# B&R Automation Studio project PT_KB_V01 (part 9)

#### Cyclic.st - Cyclic code
```iecst
PROGRAM _CYCLIC
	(* ======================================================================== *)
	(* Rad_PG_KB_CYCLIC                                                          *)
	(* Rad_PG_KB.Sequence.State masina izbora i rada izvora termalne vode: BRB2 (1) ili IEBKB1 (2). *)
	(* Prelazak izmedju grana ide iskljucivo preko PG_00_Stand_By - direktan     *)
	(* prelazak 1->2 ili 2->1 nije moguc.                                       *)
	(* ======================================================================== *)

	(* -------------------------------------------------------------------------- *)
	(* 1) Vracanje projektnih podrazumevanih parametara                          *)
	(* -------------------------------------------------------------------------- *)
	IF Rad_PG_KB.HMI.Cntrl.SetDefaultParameters THEN
		(* 1.1) Izlazne pumpe iza prihvatnog tanka. *)
		(* Aktivni SP zavisi od izabrane regulacije pritiska ili nivoa. *)
		PGRad.Par.SetPritisakPotisa := 1.2;
		PGRad.Par.SetPointNivoTanka := 1.5;
		PGRad.Par.SetPointNivoTankaUpozorenje := 2.1; (* Informativni prag; stvarni fizicki preliv je ~2.15-2.2 m. *)
		PGRad.Par.PocetnaFrekvencaIzlaznePumpe := 10.0;

		(* Centralne granice PID izlaza za obe pumpe iza prihvatnog tanka. *)
		PGRad.Par.MinFR_Pumpe := 10.0;
		PGRad.Par.MaxFR_Pumpe := 45.0;
		(* MinFR_Pumpe se u PID_Pu_PT propagira na PID_Pu_PT.MinOut. *)
		(* MaxFR_Pumpe se preko PGRad_Cmd.PID.MaxOut propagira na PID_Pu_PT.MaxOut. *)
		PGRad.Par.TimeSP.OverlapPumpi_s := 10.0;
		PGRad.Par.TimeSP.AutoRestartDelay_s := 60.0;

		(* 1.2) BRB2 priprema i ispiranje dovodne grane. *)
		PGRad.Par.MinProtok := 1.5; (* Rezervisano; trenutno nema izvrsnog potrosaca. *)
		PGRad.Par.MaxProtok := 16.2;
		PGRad.Par.SetPointMinTempIspiranja := 60.0;
		PGRad.Par.BRB2Preparation.MinTemperature_degC := 60.0;
		PGRad.Par.BRB2Preparation.MinFlow_lps := 3.0;
		PGRad.Par.BRB2Preparation.FlowTimeout_s := 30.0;
		PGRad.Par.BRB2Preparation.TemperatureAlarm_s := 5400.0;
		PGRad.Par.BRB2Preparation.TemperatureStopDelay_s := 900.0;
		PGRad.Par.BRB2Preparation.PressureAlarmDelay_s := 5.0;
		PGRad.Par.BRB2Preparation.PressureStopDelay_s := 8.0;

		(* 1.3) Lokalna hidraulika PV05 i ulaza u prihvatni tank. *)
		PGRad.Par.SetPointPritisakPV05Ispiranje := 5.5;
		PGRad.Par.SetPointPritisakUlazTanka := 5.5;
		PGRad.Par.SetPointMaxPritisakDolaznaCev := 6.5;
		PGRad.Par.TimeSP.PrelazPV05Cuvar_s := 15.0;
		PGRad.Par.MaxOtvorPropZaZatvaranje := 3;

		(* 1.4) Kontrolisani transfer sa IEBKB1 na BRB2. *)
		PGRad.Par.Transfer.PV05StartPressure_bar := 5.5;
		PGRad.Par.Transfer.PV05FinalPressure_bar := 6.5;
		PGRad.Par.Transfer.TankInletPressure_bar := 5.5;
		PGRad.Par.Transfer.PressureRamp_s := 15.0;
		PGRad.Par.Transfer.FlowTimeout_s := 30.0;
		PGRad.Par.Transfer.PV05ClosedPercent := 4.0;

		(* 1.5) Zajednicki nadzor ventila i procesnih interlock-a. *)
		PGRad.Par.TimeSP.ValvePositionTimeout_s := 30.0;
		PGRad.Par.TimeSP.InterlockDebounce_s := 2.0;

		(* 1.6) BRB2 odzracivanje: oba ventila, prag 1.5 bar sa 0.5 bar histerezom. *)
		PGRad.Par.AirRelease.BRB2.PV03.NumberOfLS := 2;
		PGRad.Par.AirRelease.BRB2.PV03.PressureSP_bar := 1.5;
		PGRad.Par.AirRelease.BRB2.PV03.PressureHysteresis_bar := 0.5;
		PGRad.Par.AirRelease.BRB2.PV03.LS1.SP_Percent := 20.0;
		PGRad.Par.AirRelease.BRB2.PV03.LS1.Ramp_PercentPerSecond := 2.0;
		PGRad.Par.AirRelease.BRB2.PV03.LS1.ConfirmTime_s := 1.0;
		PGRad.Par.AirRelease.BRB2.PV03.LS2.SP_Percent := 89.0;
		PGRad.Par.AirRelease.BRB2.PV03.LS2.Ramp_PercentPerSecond := 15.0;
		PGRad.Par.AirRelease.BRB2.PV03.LS2.ConfirmTime_s := 1.0;
		PGRad.Par.AirRelease.BRB2.PV04 := PGRad.Par.AirRelease.BRB2.PV03;

		(* 1.7) IEBKB1 odzracivanje: aktivan je PV03 sa nizim pragom pritiska. *)
		PGRad.Par.AirRelease.IEBKB1.PV03.NumberOfLS := 2;
		PGRad.Par.AirRelease.IEBKB1.PV03.PressureSP_bar := 0.15;
		PGRad.Par.AirRelease.IEBKB1.PV03.PressureHysteresis_bar := 0.05;
		PGRad.Par.AirRelease.IEBKB1.PV03.LS1.SP_Percent := 20.0;
		PGRad.Par.AirRelease.IEBKB1.PV03.LS1.Ramp_PercentPerSecond := 2.0;
		PGRad.Par.AirRelease.IEBKB1.PV03.LS1.ConfirmTime_s := 1.0;
		PGRad.Par.AirRelease.IEBKB1.PV03.LS2.SP_Percent := 89.0;
		PGRad.Par.AirRelease.IEBKB1.PV03.LS2.Ramp_PercentPerSecond := 15.0;
		PGRad.Par.AirRelease.IEBKB1.PV03.LS2.ConfirmTime_s := 1.0;
		PGRad.Par.AirRelease.IEBKB1.PV04 := PGRad.Par.AirRelease.IEBKB1.PV03;

		Rad_PG_KB.HMI.Cntrl.SetDefaultParameters := FALSE;
	END_IF

	(* -------------------------------------------------------------------------- *)
	(* 2) Podrazumevane neretentivne komande po scan-u                            *)
	(* -------------------------------------------------------------------------- *)
	PGRad_Cmd.Aktivan := FALSE;
	PGRad_Cmd.Ventili._03_Open := FALSE;
	PGRad_Cmd.Ventili._04_Open := FALSE;
	PGRad_Cmd.Ventili._05_Open := FALSE;
	PGRad_Cmd.Ventili._06_Open := FALSE;
	PGRad_Cmd.Ventili._07_Open := FALSE;

	PGRad_Cmd.PropVentili.PV01.Enable := FALSE;
	PGRad_Cmd.PropVentili.PV01.SP_Percent := 0.0;
	PGRad_Cmd.PropVentili.PV02.Enable := FALSE;
	PGRad_Cmd.PropVentili.PV02.SP_Percent := 0.0;
	PGRad_Cmd.PropVentili.PV05.Enable := FALSE;
	PGRad_Cmd.PropVentili.PV05.SP_Percent := 0.0;
	PGRad_Cmd.AirRelease.PV03.Enable := FALSE;
	PGRad_Cmd.AirRelease.PV04.Enable := FALSE;
	PGRad_Cmd.AirRelease.UseIEBKB1Parameters := FALSE;
	PGRad_Cmd.AirRelease.ResetAll := Rad_PG_KB.HMI.Cntrl.Reset;

	PGRad_Cmd.Pumpe._01.Run := FALSE;
	PGRad_Cmd.Pumpe._02.Run := FALSE;
	PGRad_Cmd.PID.Enable := FALSE;
	PGRad_Cmd.PID.ActValue := 0.0;
	PGRad_Cmd.PID.SetValue := 0.0;
	PGRad_Cmd.PID.Invert := FALSE;
	(* Jedinstvena maksimalna PID frekvencija ne zavisi od izabrane pumpe. *)
	PGRad_Cmd.PID.MaxOut := PGRad.Par.MaxFR_Pumpe;
	PGRad_Cmd.PID.EnableTracking := FALSE;
	(* Jedinstvena pocetna frekvencija koristi se pri ukljucenju PID tracking-a. *)
	PGRad_Cmd.PID.TrackingValue := PGRad.Par.PocetnaFrekvencaIzlaznePumpe;
	PGRad_BRB2Cmd.RadKaPodstanici := FALSE;
	PGRad_BRB2Cmd.ZahtevStarta := FALSE;
	PGRad_BRB2Cmd.ZahtevZaustavljanja := FALSE;
	PGRad_BRB2Cmd.ManualMode := Rad_PG_KB.HMI.Manual.Enable;
	PGRad_BRB2Cmd.ManualSequence := Rad_PG_KB.HMI.Manual.Sequence;
	PGRad_BRB2Cmd.ManualStart := Rad_PG_KB.HMI.Manual.Start;
	PGRad_BRB2Cmd.ManualStop := Rad_PG_KB.HMI.Manual.Stop;
	PGRad_BRB2Cmd.ManualNextStep := Rad_PG_KB.HMI.Manual.NextStep;
	PGRad_BRB2Cmd.ManualAbort := Rad_PG_KB.HMI.Manual.Abort;
	PGRad_BRB2Cmd.VentiliPodstaniceZatvoreni := FALSE;
	PGRad_BRB2Cmd.PritisakIEBKB1 := IEB_KB1.Sens.Pt.B_02._01_value;
	PGRad_BRB2Cmd.PodstanicaURezimuRada := FALSE;
	PGRad_BRB2Cmd.RegulationMode := 0;
	PGRad_BRB2Cmd.RegulationPV := 0.0;
	PGRad_BRB2Cmd.RegulationSP := 0.0;
	PGRad_BRB2Cmd.RegulationPVValid := FALSE;
	PGRad_BRB2Cmd.RegulationInvert := FALSE;
	PGRad_BRB2Cmd.NivoPrihvatniSud := NivoPrihvatniSud;
	IEB_KB1.Cntrl.Comm.Podstanica.Zahtev.ZahtevVode := FALSE;
	IEB_KB1.Cntrl.Comm.Podstanica.Zahtev.NivoPrihvatnogTanka := NivoPrihvatniSud;
	IEB_KB1.Cntrl.Comm.Podstanica.Zahtev.CiljaniProtok := PGRad.Par.MaxProtok;
	IEB_KB1.Cntrl.Comm.Podstanica.Zahtev.ModRada := 0;
	IEB_KB1.Cntrl.proba := FALSE;

	(* Izbor izvora sa HMI prihvata se samo u bezbednom Standby stanju. *)
	IF Rad_PG_KB.Sequence.State = PG_00_Stand_By THEN
		IF Rad_PG_KB.HMI.Cntrl.SelectIEBKB1 THEN
			PGRad.Ctrl.SelektovaniIzvor := _02_IEBKB1;
		ELSE
			PGRad.Ctrl.SelektovaniIzvor := _01_BRB2;
		END_IF;
	ELSE
		Rad_PG_KB.HMI.Cntrl.SelectIEBKB1 := PGRad.Ctrl.SelektovaniIzvor = _02_IEBKB1;
	END_IF;

	(* -------------------------------------------------------------------------- *)
	(* 3) Tajmeri pripreme BRB2 dovodne putanje                                  *)
	(* -------------------------------------------------------------------------- *)
	Rad_PG_KB.Timer.PG_V01.Close.IN := FALSE;
	Rad_PG_KB.Timer.PG_V01.Close.PT := REAL_TO_TIME(PGRad.Par.TimeSP.ValvePositionTimeout_s * 1000.0);
	Rad_PG_KB.Timer.PG_V02.Open.IN := FALSE;
	Rad_PG_KB.Timer.PG_V02.Open.PT := REAL_TO_TIME(PGRad.Par.TimeSP.ValvePositionTimeout_s * 1000.0);
	Rad_PG_KB.Timer.PG_V02.Close.IN := FALSE;
	Rad_PG_KB.Timer.PG_V02.Close.PT := REAL_TO_TIME(PGRad.Par.TimeSP.ValvePositionTimeout_s * 1000.0);
	Rad_PG_KB.Timer.PG_V01.Open.IN := FALSE;
	Rad_PG_KB.Timer.PG_V01.Open.PT := REAL_TO_TIME(PGRad.Par.TimeSP.ValvePositionTimeout_s * 1000.0);
	Rad_PG_KB.Timer.IEBKB1.StartProtokTimeout.IN := FALSE;
	Rad_PG_KB.Timer.IEBKB1.StartProtokTimeout.PT := REAL_TO_TIME(PGRad.Par.TimeSP.ValvePositionTimeout_s * 1000.0);
	Rad_PG_KB.Timer.IEBKB1.ProtokNula.IN := FALSE;
	Rad_PG_KB.Timer.IEBKB1.ProtokNula.PT := REAL_TO_TIME(PGRad.Par.TimeSP.InterlockDebounce_s * 1000.0);
	Rad_PG_KB.Timer.IEBKB1.StopProtokTimeout.IN := FALSE;
	Rad_PG_KB.Timer.IEBKB1.StopProtokTimeout.PT := REAL_TO_TIME(PGRad.Par.TimeSP.ValvePositionTimeout_s * 1000.0);
	Rad_PG_KB.Timer.PG_V05.Close.IN := FALSE;
	Rad_PG_KB.Timer.PG_V05.Close.PT := REAL_TO_TIME(PGRad.Par.TimeSP.ValvePositionTimeout_s * 1000.0);
	Rad_PG_KB.Timer.Transfer.PV05Guard.IN := FALSE;
	Rad_PG_KB.Timer.Transfer.PV05Guard.PT := REAL_TO_TIME(PGRad.Par.TimeSP.PrelazPV05Cuvar_s * 1000.0);
	Rad_PG_KB.Timer.BRB2.PreparationFlow.IN := FALSE;
	Rad_PG_KB.Timer.BRB2.PreparationFlow.PT := REAL_TO_TIME(PGRad.Par.BRB2Preparation.FlowTimeout_s * 1000.0);
	Rad_PG_KB.Timer.BRB2.TemperatureAlarm.IN := FALSE;
	Rad_PG_KB.Timer.BRB2.TemperatureAlarm.PT := REAL_TO_TIME(PGRad.Par.BRB2Preparation.TemperatureAlarm_s * 1000.0);
	Rad_PG_KB.Timer.BRB2.TemperatureStop.IN := FALSE;
	Rad_PG_KB.Timer.BRB2.TemperatureStop.PT := REAL_TO_TIME(PGRad.Par.BRB2Preparation.TemperatureStopDelay_s * 1000.0);
	Rad_PG_KB.Timer.BRB2.PressureAlarm.IN := FALSE;
	Rad_PG_KB.Timer.BRB2.PressureAlarm.PT := REAL_TO_TIME(PGRad.Par.BRB2Preparation.PressureAlarmDelay_s * 1000.0);
	Rad_PG_KB.Timer.BRB2.PressureStop.IN := FALSE;
	Rad_PG_KB.Timer.BRB2.PressureStop.PT := REAL_TO_TIME(PGRad.Par.BRB2Preparation.PressureStopDelay_s * 1000.0);
	Rad_PG_KB.Timer.Transfer.Flow.IN := FALSE;
	Rad_PG_KB.Timer.Transfer.Flow.PT := REAL_TO_TIME(PGRad.Par.Transfer.FlowTimeout_s * 1000.0);
	Rad_PG_KB.AutoRestart.Timer.IN := FALSE;
	Rad_PG_KB.AutoRestart.Timer.PT := REAL_TO_TIME(PGRad.Par.TimeSP.AutoRestartDelay_s * 1000.0);

	(* -------------------------------------------------------------------------- *)
	(* 3b) Informativna napomena: nivo prihvatnog suda blizu fizickog preliva.    *)
	(* Samo obavestenje za HMI, bez ikakve upravljacke akcije ili interlock-a -   *)
	(* ocekivano tokom regulacije temperature sekundara/protoka sa bunara uz      *)
	(* pritisak potisa izlazne pumpe.                                            *)
	(* -------------------------------------------------------------------------- *)
	Rad_PG_KB.Status.PrihvatniSudBlizuPreliva := NivoPrihvatniSud >= PGRad.Par.SetPointNivoTankaUpozorenje;

	(* -------------------------------------------------------------------------- *)
	(* 4) Glavna state masina izvora termalne vode                                *)
	(* -------------------------------------------------------------------------- *)
	(* Rad_PG_KB.HMI.Manual.Start grane imaju prioritet evaluacije. BRB2 auto-start je blokiran  *)
	(* sa Rad_PG_KB.HMI.Manual.Enable, dok IEBKB1 auto-start grana nema eksplicitnu tu proveru.    *)
	CASE Rad_PG_KB.Sequence.State OF

		PG_00_Stand_By:
			(* Neretentivni vektor je bezbedno resetovan u sekciji 2; V01/V02 se ne menjaju. *)
			Rad_PG_KB.Status.PV05.FlushingOpened := FALSE;
			(* Automatski start posle WARMSTART-a (nestanak struje), samo ako je operater *)
			(* aktivirao PGRad.Ctrl.AutoRestart. Prekida se ako se pojavi Fault ili se    *)
			(* rucno napusti Standby/automatski rezim u toku odlozenog starta.           *)
			Rad_PG_KB.AutoRestart.Timer.IN :=
				Rad_PG_KB.AutoRestart.WarmstartDetected
				AND PGRad.Ctrl.AutoRestart
				AND (NOT Rad_PG_KB.HMI.Manual.Enable)
				AND (NOT Rad_PG_KB.Diag.Fault.Latched)
				AND (PGRad.Ctrl.RegulacionaVarijanta <> _00_neaktivan);
			IF Rad_PG_KB.AutoRestart.Timer.Q THEN
				Rad_PG_KB.HMI.Cntrl.Start := TRUE;
				Rad_PG_KB.AutoRestart.WarmstartDetected := FALSE; (* jednokratno okidanje *)
			END_IF;
			(* Start je dozvoljen samo sa izabranim izvorom i regulacionom varijantom. *)
			IF Rad_PG_KB.HMI.Manual.Enable AND Rad_PG_KB.HMI.Manual.Start AND (Rad_PG_KB.HMI.Manual.Sequence = 1) THEN
				PGRad.Ctrl.SelektovaniIzvor := _01_BRB2;
				Rad_PG_KB.HMI.Manual.Start := FALSE;
				Rad_PG_KB.Sequence.State := PG_01_Priprema_BRB2;
				Rad_PG_KB.Sequence.Substep := 0;
			ELSIF Rad_PG_KB.HMI.Manual.Enable AND Rad_PG_KB.HMI.Manual.Start AND (Rad_PG_KB.HMI.Manual.Sequence = 2) THEN
				PGRad.Ctrl.SelektovaniIzvor := _02_IEBKB1;
				Rad_PG_KB.HMI.Manual.Start := FALSE;
				Rad_PG_KB.Sequence.State := PG_11_Priprema_IEBKB1;
				Rad_PG_KB.Sequence.Substep := 0;
			ELSIF Rad_PG_KB.HMI.Cntrl.Start
				AND (NOT Rad_PG_KB.HMI.Manual.Enable)
				AND (NOT Rad_PG_KB.Diag.Fault.Latched)
				AND (PGRad.Ctrl.RegulacionaVarijanta <> _00_neaktivan)
				AND (PGRad.Ctrl.SelektovaniIzvor = _01_BRB2) THEN
				Rad_PG_KB.Sequence.State := PG_01_Priprema_BRB2;
				Rad_PG_KB.Sequence.Substep := 0;
			ELSIF Rad_PG_KB.HMI.Cntrl.Start
				AND (NOT Rad_PG_KB.Diag.Fault.Latched)
				AND (PGRad.Ctrl.RegulacionaVarijanta <> _00_neaktivan)
				AND (PGRad.Ctrl.SelektovaniIzvor = _02_IEBKB1) THEN
				Rad_PG_KB.Sequence.State := PG_11_Priprema_IEBKB1;
				Rad_PG_KB.Sequence.Substep := 0;
			END_IF

		PG_01_Priprema_BRB2:
			IF Rad_PG_KB.HMI.Manual.Stop OR Rad_PG_KB.HMI.Manual.Abort THEN
				Rad_PG_KB.HMI.Cntrl.Stop := TRUE;
				Rad_PG_KB.HMI.Manual.Stop := FALSE;
				Rad_PG_KB.HMI.Manual.Abort := FALSE;
			END_IF;
			PGRad_BRB2Cmd.RadKaPodstanici := TRUE;
			PGRad_BRB2Cmd.ZahtevStarta := TRUE;
			CASE Rad_PG_KB.Sequence.Substep OF
				0:
					(* Prioritet BRB2: najpre zatvori dovod sa IEBKB1. *)
					PGRad.CmdRetain.V01_Open := FALSE;
					Rad_PG_KB.Sequence.Substep := 1;

				1:
					(* Otvaranje BRB2 dovoda je dozvoljeno tek po potvrdi zatvorenog V01. *)
					PGRad.CmdRetain.V01_Open := FALSE;
					Rad_PG_KB.Timer.PG_V01.Close.IN := NOT PG.Act.AV._1.Closed;
					IF PG.Act.AV._1.Closed AND (NOT Rad_PG_KB.HMI.Manual.Enable OR Rad_PG_KB.HMI.Manual.NextStep) THEN
						Rad_PG_KB.HMI.Manual.NextStep := FALSE;
						PGRad.CmdRetain.V02_Open := TRUE;
						Rad_PG_KB.Sequence.Substep := 2;
					ELSIF Rad_PG_KB.Timer.PG_V01.Close.Q THEN
						PGRad.CmdRetain.V01_Open := FALSE;
						PGRad.CmdRetain.V02_Open := FALSE;
						Rad_PG_KB.Diag.Fault.Latched := TRUE;
						Rad_PG_KB.Diag.Fault.Code := 11;
						Rad_PG_KB.Diag.Fault.Text := 'PG_V01 nije zatvoren za zadato vreme';
						Rad_PG_KB.Sequence.State := PG_00_Stand_By;
						Rad_PG_KB.Sequence.Substep := 0;
					END_IF

				2:
					(* Ceka se fizicka potvrda otvorenog BRB2 dovoda. *)
					PGRad.CmdRetain.V01_Open := FALSE;
					PGRad.CmdRetain.V02_Open := TRUE;
					Rad_PG_KB.Timer.PG_V02.Open.IN := NOT PG.Act.AV._2.Opened;
					IF PG.Act.AV._2.Opened AND (NOT Rad_PG_KB.HMI.Manual.Enable OR Rad_PG_KB.HMI.Manual.NextStep) THEN
						Rad_PG_KB.HMI.Manual.NextStep := FALSE;
						Rad_PG_KB.Sequence.Substep := 3;
					ELSIF Rad_PG_KB.Timer.PG_V02.Open.Q THEN
						PGRad.CmdRetain.V01_Open := FALSE;
						PGRad.CmdRetain.V02_Open := FALSE;
						Rad_PG_KB.Diag.Fault.Latched := TRUE;
						Rad_PG_KB.Diag.Fault.Code := 12;
						Rad_PG_KB.Diag.Fault.Text := 'PG_V02 nije otvoren za zadato vreme';
						Rad_PG_KB.Sequence.State := PG_00_Stand_By;
						Rad_PG_KB.Sequence.Substep := 0;
					END_IF

				3:
					(* PG_PV05 se otvara nakon dostignutog PT06 pritiska; temperatura se proverava tek posle BRB2 minimuma. *)
					IF PG.Sens.Pt._6.AI_Output.ScaledValue >= PGRad.Par.SetPointPritisakPV05Ispiranje THEN
						Rad_PG_KB.Status.PV05.FlushingOpened := TRUE;
					END_IF;
					IF Rad_PG_KB.Status.PV05.FlushingOpened THEN
						PGRad_Cmd.Aktivan := TRUE;
						PGRad_Cmd.PropVentili.PV05.Enable := TRUE;
					END_IF;
					IF PGRad_BRB2.IspiranjeMinTrajanjeDostignuto
						AND (PG.Sens.Tt._7.AI_Output.ScaledValue >= PGRad.Par.SetPointMinTempIspiranja) THEN
						IF Rad_PG_KB.HMI.Manual.Enable AND NOT Rad_PG_KB.HMI.Manual.NextStep THEN
							(* Manual mode holds the completed rinse step until operator confirmation. *)
						ELSE
							Rad_PG_KB.HMI.Manual.NextStep := FALSE;
							IF Rad_PG_KB.HMI.Manual.Enable AND (Rad_PG_KB.HMI.Manual.Sequence = 1) THEN
								(* Manual flush ends here; controlled stop closes the BRB2 path. *)
								Rad_PG_KB.HMI.Cntrl.Stop := TRUE;
								Rad_PG_KB.Sequence.State := PG_03_Zaustavljanje_BRB2;
								Rad_PG_KB.Sequence.Substep := 0;
							ELSE
								Rad_PG_KB.Sequence.Substep := 4;
							END_IF
						END_IF
					END_IF

				4:
					(* Priprema puta ka tanku: otvara se samo ON/OFF ventil izabranog ulaznog PV-a. *)
					PGRad_Cmd.Aktivan := TRUE;
					PGRad_Cmd.PropVentili.PV05.Enable := TRUE;
					CASE PGRad.Ctrl.AktivniPropVentilUlazTanka OF
						_01_PG_PV01, _02_PG_PV02:
							Rad_PG_KB.Sequence.Substep := 5;
					END_CASE

				5:
					(* Mek prelaz: ulazni PV vodi PT04, a PT06 SP PG_PV05 raste 5.5 -> 6.5 bar. *)
					PGRad_Cmd.Aktivan := TRUE;
					PGRad_Cmd.PropVentili.PV05.Enable := TRUE;
					Rad_PG_KB.Timer.Transfer.PV05Guard.IN := TRUE;
					IF Rad_PG_KB.Timer.Transfer.PV05Guard.Q AND (NOT Rad_PG_KB.HMI.Manual.Enable OR Rad_PG_KB.HMI.Manual.NextStep) THEN
						Rad_PG_KB.HMI.Manual.NextStep := FALSE;
						Rad_PG_KB.Sequence.Substep := 6;
					END_IF

				6:
					(* Punjenje tanka: PV05 je cuvar PT06, a aktivni ulazni PV odrzava PT04. *)
					PGRad_Cmd.Aktivan := TRUE;
					PGRad_Cmd.PropVentili.PV05.Enable := TRUE;
					IF (NivoPrihvatniSud >= PGRad.Par.SetPointNivoTanka)
						AND (NOT Rad_PG_KB.HMI.Manual.Enable OR Rad_PG_KB.HMI.Manual.NextStep) THEN
						Rad_PG_KB.HMI.Manual.NextStep := FALSE;
						Rad_PG_KB.Sequence.State := PG_02_Rad_BRB2;
						Rad_PG_KB.Sequence.Substep := 0;
					END_IF

			ELSE
				Rad_PG_KB.Sequence.Substep := 0;
			END_CASE

		PG_02_Rad_BRB2:
			PGRad_BRB2Cmd.RadKaPodstanici := TRUE;
			PGRad_BRB2Cmd.ZahtevStarta := TRUE;
			(* Podstanica bira aktivni BRB2 PV/SP; BRB2 lokalno menja samo FR_set. *)
			CASE PGRad.Ctrl.BRB2Regulacija OF
				BRB2_01_REG_PROTOK:
					PGRad_BRB2Cmd.RegulationMode := 1;
					PGRad_BRB2Cmd.RegulationPV := PG.Sens.MP._1.AI_Output.ScaledValue;
					PGRad_BRB2Cmd.RegulationSP := PGRad.Par.MaxProtok;
					PGRad_BRB2Cmd.RegulationPVValid := PG.Sens.MP._1.AI_Output.Status;
				BRB2_02_REG_NIVO:
					PGRad_BRB2Cmd.RegulationMode := 2;
					PGRad_BRB2Cmd.RegulationPV := NivoPrihvatniSud;
					PGRad_BRB2Cmd.RegulationSP := PGRad.Par.SetPointNivoTanka;
					PGRad_BRB2Cmd.RegulationPVValid :=
						PG.Sens.Pt._NS1.AI_Output.Status
						AND PG.Sens.Pt._NS2.AI_Output.Status;
				BRB2_03_REG_TEMPERATURA:
					PGRad_BRB2Cmd.RegulationMode := 3;
					PGRad_BRB2Cmd.RegulationPV := PG01_Local.PGSens.Tt09.Value;
					PGRad_BRB2Cmd.RegulationSP := PGRad.Par.SetPointMinTempIspiranja;
					PGRad_BRB2Cmd.RegulationPVValid := PG01_Local.PGSens.Tt09.Valid;
			END_CASE
			(* Odrzava PID regulaciju ulaza i PT06 cuvara nakon punjenja tanka. *)
			PGRad_Cmd.Aktivan := TRUE;
			PGRad_Cmd.PropVentili.PV05.Enable := TRUE;

			(* Izlaznu pumpu pokrece i frekvencu vodi iskljucivo PID_Pu_PT. *)
			PGRad_Cmd.PID.Enable :=
				(PGRad.Ctrl.RegulacionaVarijanta = _01_REG_PRITISAK)
				OR (PGRad.Ctrl.RegulacionaVarijanta = _02_REG_NIVO);

			IF PGRad_Cmd.PID.Enable THEN
				PGRad_Cmd.PID.EnableTracking := (Rad_PG_KB.Sequence.Substep = 0);
				Rad_PG_KB.Sequence.Substep := 1;
			END_IF

			(* BRB2 sme preci u rad tek kada je tank pun i izabrana PG pumpa stvarno radi. *)
			PGRad_BRB2Cmd.PodstanicaURezimuRada :=
				(NivoPrihvatniSud >= PGRad.Par.SetPointNivoTanka)
				AND (
					((PGRad.Ctrl.AktivnaPumpaIzlazTanka = _01_Pu_PG_01)
						AND PG.Act.Pu._1.Status_inRun)
					OR ((PGRad.Ctrl.AktivnaPumpaIzlazTanka = _02_Pu_PG_02)
						AND PG.Act.Pu._2.Status_inRun)
				);

			(* Napusta granu cim PGRad.Ctrl.SelektovaniIzvor vise nije _01_BRB2. *)
			IF Rad_PG_KB.HMI.Cntrl.Stop OR (PGRad.Ctrl.SelektovaniIzvor <> _01_BRB2) THEN
				Rad_PG_KB.Sequence.State := PG_03_Zaustavljanje_BRB2;
				Rad_PG_KB.Sequence.Substep := 0;
			END_IF

		PG_03_Zaustavljanje_BRB2:
			(* PT najpre trazi BRB2 ramp-down, zatim zatvara PV grane po stop SP potvrdi. *)
			PGRad_Cmd.Aktivan := TRUE;
			PGRad_BRB2Cmd.ZahtevZaustavljanja := TRUE;

			IF Rad_PG_KB.Sequence.Substep = 0 THEN
				Rad_PG_KB.Status.Pump.OutletStopped := TRUE;
				Rad_PG_KB.Sequence.Substep := 1;
			END_IF;

			(* Izlazna pumpa ostaje na aktivnoj regulaciji dok tank ne padne ispod 60% SP-a. *)
			IF NivoPrihvatniSud < (0.6 * PGRad.Par.SetPointNivoTanka) THEN
				Rad_PG_KB.Status.Pump.OutletStopped := FALSE;
			END_IF;

			IF Rad_PG_KB.Status.Pump.OutletStopped THEN
				PGRad_Cmd.PID.Enable :=
					(PGRad.Ctrl.RegulacionaVarijanta = _01_REG_PRITISAK)
					OR (PGRad.Ctrl.RegulacionaVarijanta = _02_REG_NIVO);
			END_IF;

			(* Izlazni ventil ostaje otvoren dok ATV ne potvrdi da se pumpa zaustavila. *)
			IF NOT Rad_PG_KB.Status.Pump.OutletStopped THEN
				CASE PGRad.Ctrl.AktivnaPumpaIzlazTanka OF
					_01_Pu_PG_01:
						PGRad_Cmd.Ventili._03_Open := PG.Act.Pu._1.Status_inRun;
					_02_Pu_PG_02:
						PGRad_Cmd.Ventili._04_Open := PG.Act.Pu._2.Status_inRun;
				END_CASE
			END_IF;

			IF NOT PGRad_BRB2.StopSPDostignut THEN
				(* Dok BRB2 spusta frekvenciju, PT06 i PT04 ostaju u regulaciji. *)
				PGRad_Cmd.PropVentili.PV05.Enable := TRUE;
			END_IF;

			(* Nakon BRB2 stop SP-a svi proporcionalni ventili ostaju bez zahteva. *)
			PGRad_BRB2Cmd.VentiliPodstaniceZatvoreni := PGRad_BRB2.StopSPDostignut
				AND (PG.Act.PV._1.PV_Output.PV_Percent <= PGRad.Par.MaxOtvorPropZaZatvaranje)
				AND (PG.Act.PV._2.PV_Output.PV_Percent <= PGRad.Par.MaxOtvorPropZaZatvaranje)
				AND (PG.Act.PV._5.PV_Output.PV_Percent <= PGRad.Par.MaxOtvorPropZaZatvaranje);

			IF PGRad_BRB2.RB2V02Zatvoren
				AND NOT Rad_PG_KB.Status.Pump.OutletStopped
				AND NOT PG.Act.Pu._1.Status_inRun
				AND NOT PG.Act.Pu._2.Status_inRun THEN
				Rad_PG_KB.Sequence.State := PG_00_Stand_By;
				Rad_PG_KB.Sequence.Substep := 0;
			END_IF

		PG_11_Priprema_IEBKB1:
			(* IEBKB1 put koristi samo PG_V01 i PG_V05; PV01/PV02/V06/V07 ostaju zatvoreni. *)
			IEB_KB1.Cntrl.Comm.Podstanica.Zahtev.ZahtevVode := TRUE;
			IEB_KB1.Cntrl.Comm.Podstanica.Zahtev.ModRada := 1;
			IEB_KB1.Cntrl.proba := TRUE;
			CASE Rad_PG_KB.Sequence.Substep OF
				0:
					(* Najpre se opoziva zahtev otvaranja BRB2 dovoda PG_V02. *)
					PGRad.CmdRetain.V02_Open := FALSE;
					Rad_PG_KB.Sequence.Substep := 1;

				1:
					(* Ceka se zatvoren PG_V02, pa se dozvoljava otvaranje IEBKB1 dovoda PG_V01. *)
					PGRad.CmdRetain.V02_Open := FALSE;
					Rad_PG_KB.Timer.PG_V02.Close.IN := NOT PG.Act.AV._2.Closed;
					IF PG.Act.AV._2.Closed THEN
						PGRad.CmdRetain.V01_Open := TRUE;
						Rad_PG_KB.Sequence.Substep := 2;
					ELSIF Rad_PG_KB.Timer.PG_V02.Close.Q THEN
						PGRad.CmdRetain.V01_Open := FALSE;
						PGRad.CmdRetain.V02_Open := FALSE;
						Rad_PG_KB.Diag.Fault.Latched := TRUE;
						Rad_PG_KB.Diag.Fault.Code := 13;
						Rad_PG_KB.Diag.Fault.Text := 'PG_V02 nije zatvoren za zadato vreme';
						Rad_PG_KB.Sequence.State := PG_00_Stand_By;
						Rad_PG_KB.Sequence.Substep := 0;
					END_IF

				2:
					(* Ceka se fizicka potvrda otvorenog PG_V01 za IEBKB1 dovod. *)
					PGRad.CmdRetain.V01_Open := TRUE;
					PGRad.CmdRetain.V02_Open := FALSE;
					Rad_PG_KB.Timer.PG_V01.Open.IN := NOT PG.Act.AV._1.Opened;
					IF PG.Act.AV._1.Opened THEN
						Rad_PG_KB.Sequence.Substep := 3;
					ELSIF Rad_PG_KB.Timer.PG_V01.Open.Q THEN
						PGRad.CmdRetain.V01_Open := FALSE;
						Rad_PG_KB.Diag.Fault.Latched := TRUE;
						Rad_PG_KB.Diag.Fault.Code := 14;
						Rad_PG_KB.Diag.Fault.Text := 'PG_V01 nije otvoren za zadato vreme';
						Rad_PG_KB.Sequence.State := PG_00_Stand_By;
						Rad_PG_KB.Sequence.Substep := 0;
					END_IF

				3:
					(* V05 vodi IEBKB1 vodu direktno u prihvatni tank. *)
					PGRad_Cmd.Aktivan := TRUE;
					PGRad_Cmd.Ventili._05_Open := TRUE;
					Rad_PG_KB.Timer.IEBKB1.StartProtokTimeout.IN :=
						IEB_KB1.Cntrl.Comm.Podstanica.Status.TrenutniProtok <= 0.1;
					IF IEB_KB1.Cntrl.Comm.Podstanica.Status.TrenutniProtok > 0.1 THEN
						Rad_PG_KB.Sequence.Substep := 4;
					ELSIF Rad_PG_KB.Timer.IEBKB1.StartProtokTimeout.Q THEN
						Rad_PG_KB.Diag.Fault.Latched := TRUE;
						Rad_PG_KB.Diag.Fault.Code := 18;
						Rad_PG_KB.Diag.Fault.Text := 'IEBKB1 dotok nije poceo za zadato vreme';
						Rad_PG_KB.Sequence.State := PG_13_Zaustavljanje_IEBKB1;
						Rad_PG_KB.Sequence.Substep := 0;
					END_IF

				4:
					(* PG_V05 ostaje otvoren dok prihvatni tank ne dostigne zadati nivo. *)
					PGRad_Cmd.Aktivan := TRUE;
					PGRad_Cmd.Ventili._05_Open := TRUE;
					IF NivoPrihvatniSud >= PGRad.Par.SetPointNivoTanka THEN
						Rad_PG_KB.Sequence.State := PG_12_Rad_IEBKB1;
						Rad_PG_KB.Sequence.Substep := 0;
					END_IF

			ELSE
				Rad_PG_KB.Sequence.Substep := 0;
			END_CASE

		PG_12_Rad_IEBKB1:
			(* IEBKB1 dovod ostaje otvoren; PT lokalno vodi samo izlaznu pumpu. *)
			PGRad.CmdRetain.V01_Open := TRUE;
			PGRad.CmdRetain.V02_Open := FALSE;
			PGRad_Cmd.Aktivan := TRUE;
			PGRad_Cmd.Ventili._05_Open := TRUE;
			IEB_KB1.Cntrl.Comm.Podstanica.Zahtev.ZahtevVode := TRUE;
			IEB_KB1.Cntrl.Comm.Podstanica.Zahtev.ModRada := 2;
			IEB_KB1.Cntrl.proba := TRUE;

			PGRad_Cmd.PID.Enable :=
				(PGRad.Ctrl.RegulacionaVarijanta = _01_REG_PRITISAK)
				OR (PGRad.Ctrl.RegulacionaVarijanta = _02_REG_NIVO);

			IF PGRad_Cmd.PID.Enable THEN
				PGRad_Cmd.PID.EnableTracking := (Rad_PG_KB.Sequence.Substep = 0);
				Rad_PG_KB.Sequence.Substep := 1;
			END_IF

			IF Rad_PG_KB.HMI.Cntrl.Stop OR (PGRad.Ctrl.SelektovaniIzvor <> _02_IEBKB1) THEN
				Rad_PG_KB.Sequence.State := PG_13_Zaustavljanje_IEBKB1;
				Rad_PG_KB.Sequence.Substep := 0;
			ELSIF Rad_PG_KB.HMI.Cntrl.TransferToBRB2 THEN
				Rad_PG_KB.HMI.Cntrl.TransferToBRB2 := FALSE;
				IF Rad_PG_KB.Sequence.BRB2.Ready
					AND PGRad_IEBKB1Prepared.Enable
					AND PGRad_IEBKB1Prepared.InterfaceReady
					AND PGRad_IEBKB1Prepared.CommValid
					AND PGRad_IEBKB1Prepared.HeartbeatValid
					AND NOT PGRad_IEBKB1Prepared.Fault THEN
					Rad_PG_KB.Sequence.Transfer.Requested := TRUE;
					Rad_PG_KB.Sequence.State := PG_14_Transfer_IEBKB1_BRB2;
					Rad_PG_KB.Sequence.Substep := 0;
				END_IF
			END_IF

		PG_14_Transfer_IEBKB1_BRB2:
			(* Transfer je dozvoljen samo uz kompletan buduci IEBKB1 statusni ugovor. *)
			PGRad_BRB2Cmd.RadKaPodstanici := TRUE;
			PGRad_BRB2Cmd.ZahtevStarta := TRUE;
			IEB_KB1.Cntrl.Comm.Podstanica.Zahtev.ModRada := 3;
			CASE Rad_PG_KB.Sequence.Substep OF
				0:
					(* IEBKB1 zahtev vode je opozvan; PG_V05 ostaje otvoren do nultog protoka. *)
					PGRad.CmdRetain.V01_Open := TRUE;
					PGRad.CmdRetain.V02_Open := FALSE;
					PGRad_Cmd.Aktivan := TRUE;
					PGRad_Cmd.Ventili._05_Open := TRUE;
					Rad_PG_KB.Timer.IEBKB1.ProtokNula.IN := IEB_KB1.Sens.MP.B_01._01_value < 0.1;
					Rad_PG_KB.Timer.IEBKB1.StopProtokTimeout.IN := NOT Rad_PG_KB.Timer.IEBKB1.ProtokNula.Q;
					IF Rad_PG_KB.Timer.IEBKB1.ProtokNula.Q THEN
						Rad_PG_KB.Sequence.Substep := 1;
					ELSIF Rad_PG_KB.Timer.IEBKB1.StopProtokTimeout.Q THEN
						Rad_PG_KB.Diag.Fault.Latched := TRUE;
						Rad_PG_KB.Diag.Fault.Code := 31;
						Rad_PG_KB.Diag.Fault.Text := 'Transfer: IEBKB1 protok nije pao na nulu';
						Rad_PG_KB.Sequence.State := PG_13_Zaustavljanje_IEBKB1;
						Rad_PG_KB.Sequence.Substep := 1;
					END_IF

				1:
					(* Pneumatski PG_V05 se zatvara pre izolovanja IEBKB1 dovoda. *)
					PGRad.CmdRetain.V01_Open := TRUE;
					PGRad.CmdRetain.V02_Open := FALSE;
					Rad_PG_KB.Timer.PG_V05.Close.IN := NOT PG.Act.AV._5.Closed;
					IF PG.Act.AV._5.Closed THEN
						Rad_PG_KB.Sequence.Substep := 2;
					ELSIF Rad_PG_KB.Timer.PG_V05.Close.Q THEN
						Rad_PG_KB.Diag.Fault.Latched := TRUE;
						Rad_PG_KB.Diag.Fault.Code := 32;
						Rad_PG_KB.Diag.Fault.Text := 'Transfer: PG_V05 nije zatvoren';
						Rad_PG_KB.Sequence.State := PG_13_Zaustavljanje_IEBKB1;
						Rad_PG_KB.Sequence.Substep := 2;
					END_IF

				2:
					(* Tek posle zatvorenog PG_V05 zatvara se elektromotorni PG_V01. *)
					PGRad.CmdRetain.V01_Open := FALSE;
					PGRad.CmdRetain.V02_Open := FALSE;
					Rad_PG_KB.Timer.PG_V01.Close.IN := NOT PG.Act.AV._1.Closed;
					IF PG.Act.AV._1.Closed THEN
						Rad_PG_KB.Sequence.Substep := 3;
					ELSIF Rad_PG_KB.Timer.PG_V01.Close.Q THEN
						Rad_PG_KB.Diag.Fault.Latched := TRUE;
						Rad_PG_KB.Diag.Fault.Code := 33;
						Rad_PG_KB.Diag.Fault.Text := 'Transfer: PG_V01 nije zatvoren';
						Rad_PG_KB.Sequence.State := PG_13_Zaustavljanje_IEBKB1;
						Rad_PG_KB.Sequence.Substep := 3;
					END_IF

				3:
					(* PG_V02 se otvara samo uz fizicku potvrdu zatvorenog PG_V01. *)
					PGRad.CmdRetain.V01_Open := FALSE;
					PGRad.CmdRetain.V02_Open := TRUE;
					Rad_PG_KB.Timer.PG_V02.Open.IN := NOT PG.Act.AV._2.Opened;
					IF PG.Act.AV._2.Opened THEN
						Rad_PG_KB.Sequence.Substep := 4;
					ELSIF Rad_PG_KB.Timer.PG_V02.Open.Q THEN
						Rad_PG_KB.Diag.Fault.Latched := TRUE;
						Rad_PG_KB.Diag.Fault.Code := 34;
						Rad_PG_KB.Diag.Fault.Text := 'Transfer: PG_V02 nije otvoren';
						Rad_PG_KB.Sequence.State := PG_03_Zaustavljanje_BRB2;
						Rad_PG_KB.Sequence.Substep := 0;
					END_IF

				4:
					(* Dve petlje rade istovremeno: PV05/PT06 rampa i PV01/02/PT04 na 5.5 bar. *)
					PGRad_Cmd.Aktivan := TRUE;
					PGRad_Cmd.PropVentili.PV05.Enable := TRUE;
					Rad_PG_KB.Timer.Transfer.PV05Guard.IN := TRUE;
					Rad_PG_KB.Timer.Transfer.Flow.IN := NOT PGRad_BRB2.IspiranjeProtokDostignut;
					IF Rad_PG_KB.Timer.Transfer.Flow.Q THEN
						Rad_PG_KB.Diag.Fault.Latched := TRUE;
						Rad_PG_KB.Diag.Fault.Code := 35;
						Rad_PG_KB.Diag.Fault.Text := 'Transfer: BRB2 protok nije potvrden';
						Rad_PG_KB.Sequence.State := PG_03_Zaustavljanje_BRB2;
						Rad_PG_KB.Sequence.Substep := 0;
					ELSIF Rad_PG_KB.Timer.Transfer.PV05Guard.Q
						AND PGRad_BRB2.IspiranjeProtokDostignut
						AND (PG.Act.PV._5.PV_Output.PV_Percent <= PGRad.Par.Transfer.PV05ClosedPercent) THEN
						Rad_PG_KB.Sequence.Transfer.Requested := FALSE;
						Rad_PG_KB.Sequence.BRB2.PreparationState := BRB2_PREP_00_IDLE;
						Rad_PG_KB.Sequence.State := PG_02_Rad_BRB2;
						Rad_PG_KB.Sequence.Substep := 0;
					END_IF

			ELSE
				Rad_PG_KB.Sequence.Substep := 0;
			END_CASE

		PG_13_Zaustavljanje_IEBKB1:
			(* ==================================================================== *)
			(* 1) Podrazumevane komande za kontrolisano zaustavljanje IEBKB1       *)
			(* ==================================================================== *)
			(* Zahtev bunaru je uklonjen; V05 ostaje otvoren do potvrdenog nultog protoka. *)
			PGRad_Cmd.Aktivan := TRUE;
			PGRad.CmdRetain.V02_Open := FALSE;
			IEB_KB1.Cntrl.Comm.Podstanica.Zahtev.ModRada := 3;
			IEB_KB1.Cntrl.proba := FALSE;

			(* ==================================================================== *)
			(* 2) Zadrzavanje rada izlazne pumpe dok se tank ne isprazni            *)
			(* ==================================================================== *)
			IF Rad_PG_KB.Sequence.Substep = 0 THEN
				Rad_PG_KB.Status.Pump.OutletStopped := TRUE;
				Rad_PG_KB.Sequence.Substep := 1;
			END_IF;

			IF NivoPrihvatniSud < (0.6 * PGRad.Par.SetPointNivoTanka) THEN
				Rad_PG_KB.Status.Pump.OutletStopped := FALSE;
			END_IF;

			IF Rad_PG_KB.Status.Pump.OutletStopped THEN
				PGRad_Cmd.PID.Enable :=
					(PGRad.Ctrl.RegulacionaVarijanta = _01_REG_PRITISAK)
					OR (PGRad.Ctrl.RegulacionaVarijanta = _02_REG_NIVO);
			END_IF

			(* Izlazni ventil ostaje otvoren dok ATV ne potvrdi da se pumpa zaustavila. *)
			IF NOT Rad_PG_KB.Status.Pump.OutletStopped THEN
				CASE PGRad.Ctrl.AktivnaPumpaIzlazTanka OF
					_01_Pu_PG_01:
						PGRad_Cmd.Ventili._03_Open := PG.Act.Pu._1.Status_inRun;
					_02_Pu_PG_02:
						PGRad_Cmd.Ventili._04_Open := PG.Act.Pu._2.Status_inRun;
				END_CASE
			END_IF

			(* ==================================================================== *)
			(* 3) Stop podkoraci: nulti protok, PG_V05, zatim PG_V01                *)
			(* ==================================================================== *)
			CASE Rad_PG_KB.Sequence.Substep OF
				1:
					PGRad.CmdRetain.V01_Open := TRUE;
					PGRad_Cmd.Ventili._05_Open := TRUE;
					Rad_PG_KB.Timer.IEBKB1.ProtokNula.IN := IEB_KB1.Sens.MP.B_01._01_value < 0.1;
					Rad_PG_KB.Timer.IEBKB1.StopProtokTimeout.IN := NOT Rad_PG_KB.Timer.IEBKB1.ProtokNula.Q;
					IF Rad_PG_KB.Timer.IEBKB1.ProtokNula.Q THEN
						Rad_PG_KB.Sequence.Substep := 2;
					ELSIF Rad_PG_KB.Timer.IEBKB1.StopProtokTimeout.Q THEN
						Rad_PG_KB.Diag.Fault.Latched := TRUE;
						Rad_PG_KB.Diag.Fault.Code := 16;
						Rad_PG_KB.Diag.Fault.Text := 'IEBKB1 dotok nije prestao za zadato vreme';
					END_IF

				2:
					(* PG_V05 se zatvara tek nakon stabilne potvrde nultog dotoka. *)
					Rad_PG_KB.Timer.PG_V05.Close.IN := NOT PG.Act.AV._5.Closed;
					IF PG.Act.AV._5.Closed THEN
						IF PGRad.Ctrl.SelektovaniIzvor = _02_IEBKB1 THEN
							IF NOT Rad_PG_KB.Status.Pump.OutletStopped
								AND NOT PG.Act.Pu._1.Status_inRun
								AND NOT PG.Act.Pu._2.Status_inRun THEN
								Rad_PG_KB.Sequence.State := PG_00_Stand_By;
								Rad_PG_KB.Sequence.Substep := 0;
							END_IF
						ELSE
							PGRad.CmdRetain.V01_Open := FALSE;
							Rad_PG_KB.Sequence.Substep := 3;
						END_IF
					ELSIF Rad_PG_KB.Timer.PG_V05.Close.Q THEN
						Rad_PG_KB.Diag.Fault.Latched := TRUE;
						Rad_PG_KB.Diag.Fault.Code := 17;
						Rad_PG_KB.Diag.Fault.Text := 'PG_V05 nije zatvoren za zadato vreme';
					END_IF

				3:
					(* V01 se zatvara samo kada je zadrzani izbor izvora promenjen. *)
					PGRad.CmdRetain.V01_Open := FALSE;
					Rad_PG_KB.Timer.PG_V01.Close.IN := NOT PG.Act.AV._1.Closed;
					IF PG.Act.AV._1.Closed
						AND NOT Rad_PG_KB.Status.Pump.OutletStopped
						AND NOT PG.Act.Pu._1.Status_inRun
						AND NOT PG.Act.Pu._2.Status_inRun THEN
						Rad_PG_KB.Sequence.State := PG_00_Stand_By;
						Rad_PG_KB.Sequence.Substep := 0;
					ELSIF Rad_PG_KB.Timer.PG_V01.Close.Q THEN
						Rad_PG_KB.Diag.Fault.Latched := TRUE;
						Rad_PG_KB.Diag.Fault.Code := 15;
						Rad_PG_KB.Diag.Fault.Text := 'PG_V01 nije zatvoren za zadato vreme';
					END_IF

			ELSE
				Rad_PG_KB.Sequence.Substep := 0;
			END_CASE

	ELSE
		(* Nepoznato stanje - bezbedan povratak na Stand_By. *)
		Rad_PG_KB.Sequence.State := PG_00_Stand_By;

	END_CASE

	(* -------------------------------------------------------------------------- *)
	(* 4.1) Centralno mapiranje PID regulacije izlazne pumpe                      *)
	(* -------------------------------------------------------------------------- *)
	(* Aktivno stanje odredjuje Enable, a izbori jedinstveno mapiraju PID i pumpu. *)
	IF PGRad_Cmd.PID.Enable THEN
		CASE PGRad.Ctrl.RegulacionaVarijanta OF
			_01_REG_PRITISAK:
				PGRad_Cmd.PID.ActValue := PG.Sens.Pt._5.AI_Output.ScaledValue;
				PGRad_Cmd.PID.SetValue := PGRad.Par.SetPritisakPotisa;
				PGRad_Cmd.PID.Invert := FALSE;

			_02_REG_NIVO:
				PGRad_Cmd.PID.ActValue := NivoPrihvatniSud;
				PGRad_Cmd.PID.SetValue := PGRad.Par.SetPointNivoTanka;
				PGRad_Cmd.PID.Invert := TRUE;
		END_CASE

		CASE PGRad.Ctrl.AktivnaPumpaIzlazTanka OF
			_01_Pu_PG_01:
				PGRad_Cmd.Ventili._03_Open := TRUE;
				PGRad_Cmd.Pumpe._01.Run := TRUE;

			_02_Pu_PG_02:
				PGRad_Cmd.Ventili._04_Open := TRUE;
				PGRad_Cmd.Pumpe._02.Run := TRUE;
		END_CASE
	END_IF

	(* -------------------------------------------------------------------------- *)
	(* 5) Nezavisna priprema BRB2 uz aktivno snabdevanje IEBKB1                   *)
	(* -------------------------------------------------------------------------- *)
	IF (Rad_PG_KB.Sequence.State = PG_12_Rad_IEBKB1) AND Rad_PG_KB.HMI.Cntrl.PrepareBRB2
		AND (Rad_PG_KB.Sequence.BRB2.PreparationState = BRB2_PREP_00_IDLE) THEN
		Rad_PG_KB.HMI.Cntrl.PrepareBRB2 := FALSE;
		Rad_PG_KB.Sequence.BRB2.Ready := FALSE;
		Rad_PG_KB.Sequence.BRB2.PreparationSubstep := 0;
		Rad_PG_KB.Sequence.BRB2.PreparationState := BRB2_PREP_10_START;
	END_IF;

	CASE Rad_PG_KB.Sequence.BRB2.PreparationState OF
		BRB2_PREP_00_IDLE:
			Rad_PG_KB.Sequence.BRB2.Ready := FALSE;

		BRB2_PREP_10_START:
			(* BRB2 startuje ka drenažnoj grani; PG_V02 ostaje zatvoren uz aktivan IEBKB1. *)
			PGRad_BRB2Cmd.RadKaPodstanici := TRUE;
			PGRad_BRB2Cmd.ZahtevStarta := TRUE;
			PGRad_Cmd.Aktivan := TRUE;
			PGRad_Cmd.PropVentili.PV05.Enable := TRUE;
			Rad_PG_KB.Timer.BRB2.PreparationFlow.IN := NOT PGRad_BRB2.IspiranjeProtokDostignut;
			IF PGRad_BRB2.PumpaAktivna AND PGRad_BRB2.IspiranjeProtokDostignut THEN
				Rad_PG_KB.Sequence.BRB2.PreparationState := BRB2_PREP_20_ZAGREVANJE;
			ELSIF Rad_PG_KB.Timer.BRB2.PreparationFlow.Q THEN
				Rad_PG_KB.Diag.Fault.Latched := TRUE;
				Rad_PG_KB.Diag.Fault.Code := 21;
				Rad_PG_KB.Diag.Fault.Text := 'BRB2 priprema: protok nije potvrden';
				Rad_PG_KB.Sequence.BRB2.PreparationState := BRB2_PREP_40_STOPPING;
			END_IF

		BRB2_PREP_20_ZAGREVANJE:
			(* IEBKB1 i dalje puni tank; BRB2 odrzava protok i zagreva vod ka PG_PV05. *)
			PGRad_BRB2Cmd.RadKaPodstanici := TRUE;
			PGRad_BRB2Cmd.ZahtevStarta := TRUE;
			PGRad_Cmd.Aktivan := TRUE;
			PGRad_Cmd.PropVentili.PV05.Enable := TRUE;
			Rad_PG_KB.Timer.BRB2.TemperatureAlarm.IN :=
				PG.Sens.Tt._7.AI_Output.ScaledValue < PGRad.Par.BRB2Preparation.MinTemperature_degC;
			Rad_PG_KB.Timer.BRB2.TemperatureStop.IN := Rad_PG_KB.Timer.BRB2.TemperatureAlarm.Q;
			IF PGRad_BRB2.IspiranjeMinTrajanjeDostignuto
				AND PGRad_BRB2.IspiranjeProtokDostignut
				AND ((PG.Sens.Tt._7.AI_Output.ScaledValue >= PGRad.Par.BRB2Preparation.MinTemperature_degC)
					OR Rad_PG_KB.HMI.Cntrl.Continue) THEN
				Rad_PG_KB.HMI.Cntrl.Continue := FALSE;
				Rad_PG_KB.Sequence.BRB2.Ready := TRUE;
				Rad_PG_KB.Sequence.BRB2.PreparationState := BRB2_PREP_30_SPReady;
			ELSIF Rad_PG_KB.Timer.BRB2.TemperatureAlarm.Q THEN
				Rad_PG_KB.Diag.Fault.Latched := TRUE;
				Rad_PG_KB.Diag.Fault.Code := 22;
				Rad_PG_KB.Diag.Fault.Text := 'BRB2 priprema: temperatura nije dostignuta';
				IF Rad_PG_KB.Timer.BRB2.TemperatureStop.Q THEN
					Rad_PG_KB.Sequence.BRB2.PreparationState := BRB2_PREP_40_STOPPING;
				END_IF
			END_IF

		BRB2_PREP_30_SPReady:
			(* Spreman BRB2 ostaje na drenaži do transfera ili kontrolisanog stopa. *)
			Rad_PG_KB.Sequence.BRB2.Ready := TRUE;
			PGRad_BRB2Cmd.RadKaPodstanici := TRUE;
			PGRad_BRB2Cmd.ZahtevStarta := TRUE;
			PGRad_Cmd.Aktivan := TRUE;
			PGRad_Cmd.PropVentili.PV05.Enable := TRUE;
			IF Rad_PG_KB.HMI.Cntrl.Stop OR Rad_PG_KB.HMI.Manual.Stop OR Rad_PG_KB.HMI.Manual.Abort THEN
				Rad_PG_KB.Sequence.BRB2.PreparationState := BRB2_PREP_40_STOPPING;
			END_IF

		BRB2_PREP_40_STOPPING, BRB2_PREP_90_FAULT:
			Rad_PG_KB.Sequence.BRB2.Ready := FALSE;
			PGRad_BRB2Cmd.ZahtevZaustavljanja := TRUE;
			PGRad_BRB2Cmd.VentiliPodstaniceZatvoreni :=
				(PG.Act.PV._1.PV_Output.PV_Percent <= PGRad.Par.MaxOtvorPropZaZatvaranje)
				AND (PG.Act.PV._2.PV_Output.PV_Percent <= PGRad.Par.MaxOtvorPropZaZatvaranje)
				AND (PG.Act.PV._5.PV_Output.PV_Percent <= PGRad.Par.MaxOtvorPropZaZatvaranje);
			IF PGRad_BRB2.RB2V02Zatvoren THEN
				Rad_PG_KB.Sequence.BRB2.PreparationState := BRB2_PREP_00_IDLE;
			END_IF
	END_CASE

	(* Visok PT06 prvo daje alarm, a tek nakon dodatnog vremena kontrolisani stop. *)
	Rad_PG_KB.Timer.BRB2.PressureAlarm.IN :=
		(Rad_PG_KB.Sequence.BRB2.PreparationState <> BRB2_PREP_00_IDLE)
		AND (PG.Sens.Pt._6.AI_Output.ScaledValue > PGRad.Par.Transfer.PV05FinalPressure_bar);
	Rad_PG_KB.Timer.BRB2.PressureStop.IN := Rad_PG_KB.Timer.BRB2.PressureAlarm.Q;
	IF Rad_PG_KB.Timer.BRB2.PressureAlarm.Q THEN
		Rad_PG_KB.Diag.Fault.Latched := TRUE;
		Rad_PG_KB.Diag.Fault.Code := 23;
		Rad_PG_KB.Diag.Fault.Text := 'BRB2 priprema: visok PT06 pritisak';
		IF Rad_PG_KB.Timer.BRB2.PressureStop.Q THEN
			Rad_PG_KB.Sequence.BRB2.PreparationState := BRB2_PREP_40_STOPPING;
		END_IF
	END_IF;

	(* Nevalidna BRB2 komunikacija ili udaljeni fault uvek vode u kontrolisani stop. *)
	IF (Rad_PG_KB.Sequence.BRB2.PreparationState <> BRB2_PREP_00_IDLE)
		AND (NOT PGRad_BRB2Watchdog.Valid OR PGRad_BRB2.BRB2Fault) THEN
		Rad_PG_KB.Sequence.BRB2.PreparationState := BRB2_PREP_40_STOPPING;
	END_IF;
	IF (Rad_PG_KB.Sequence.State = PG_02_Rad_BRB2)
		AND (NOT PGRad_BRB2Watchdog.Valid OR PGRad_BRB2.BRB2Fault) THEN
		Rad_PG_KB.Sequence.State := PG_03_Zaustavljanje_BRB2;
		Rad_PG_KB.Sequence.Substep := 0;
	END_IF;

	(* -------------------------------------------------------------------------- *)
	(* 6) Rezim rada i dozvole odzracivanja                                      *)
	(* -------------------------------------------------------------------------- *)
	(* Tokom pripreme, rada i zaustavljanja zadrzava se parametarski skup izvora. *)
	CASE Rad_PG_KB.Sequence.State OF
		PG_01_Priprema_BRB2, PG_02_Rad_BRB2, PG_03_Zaustavljanje_BRB2:
			PGRad_Cmd.AirRelease.PV03.Enable := TRUE;
			PGRad_Cmd.AirRelease.PV04.Enable := TRUE;
			PGRad_Cmd.AirRelease.UseIEBKB1Parameters := FALSE;
		PG_11_Priprema_IEBKB1, PG_12_Rad_IEBKB1, PG_13_Zaustavljanje_IEBKB1:
			PGRad_Cmd.AirRelease.PV03.Enable := TRUE;
			PGRad_Cmd.AirRelease.PV04.Enable := FALSE;
			PGRad_Cmd.AirRelease.UseIEBKB1Parameters := TRUE;
	END_CASE

	(* -------------------------------------------------------------------------- *)
	(* 7) Izvrsavanje tajmera pripreme, stop sekvence i prelaza PV05              *)
	(* -------------------------------------------------------------------------- *)
	(* IN/PT su pripremljeni u sekciji 3 i aktivnom stanju; ovde se osvezava Q/ET. *)
	Rad_PG_KB.Timer.PG_V01.Close();
	Rad_PG_KB.Timer.PG_V01.Open();
	Rad_PG_KB.Timer.PG_V02.Open();
	Rad_PG_KB.Timer.PG_V02.Close();
	Rad_PG_KB.Timer.IEBKB1.StartProtokTimeout();
	Rad_PG_KB.Timer.IEBKB1.ProtokNula();
	Rad_PG_KB.Timer.IEBKB1.StopProtokTimeout();
	Rad_PG_KB.Timer.PG_V05.Close();
	Rad_PG_KB.Timer.Transfer.PV05Guard();
	Rad_PG_KB.Timer.BRB2.PreparationFlow();
	Rad_PG_KB.Timer.BRB2.TemperatureAlarm();
	Rad_PG_KB.Timer.BRB2.TemperatureStop();
	Rad_PG_KB.Timer.BRB2.PressureAlarm();
	Rad_PG_KB.Timer.BRB2.PressureStop();
	Rad_PG_KB.Timer.Transfer.Flow();
	Rad_PG_KB.AutoRestart.Timer();

	(* -------------------------------------------------------------------------- *)
	(* 8) PID petlje proporcionalnih ventila                                     *)
	(* -------------------------------------------------------------------------- *)
	(* 8.1) PV05 cuva PT06 tokom punjenja, rada BRB2 i njegovog ramp-down-a. *)
	Rad_PG_KB.Control.PV05.PID.Enable := ((Rad_PG_KB.Sequence.State = PG_01_Priprema_BRB2) AND (Rad_PG_KB.Sequence.Substep >= 3))
		OR (Rad_PG_KB.Sequence.State = PG_02_Rad_BRB2)
		OR ((Rad_PG_KB.Sequence.State = PG_03_Zaustavljanje_BRB2) AND NOT PGRad_BRB2.StopSPDostignut)
		OR (Rad_PG_KB.Sequence.BRB2.PreparationState = BRB2_PREP_10_START)
		OR (Rad_PG_KB.Sequence.BRB2.PreparationState = BRB2_PREP_20_ZAGREVANJE)
		OR (Rad_PG_KB.Sequence.BRB2.PreparationState = BRB2_PREP_30_SPReady)
		OR ((Rad_PG_KB.Sequence.State = PG_14_Transfer_IEBKB1_BRB2) AND (Rad_PG_KB.Sequence.Substep = 4));
	Rad_PG_KB.Control.PV05.PID.ActValue := PG.Sens.Pt._6.AI_Output.ScaledValue; (* Merena vrednost PT06. *)
	(* U prelazu se SP linearno podize od ispiranja do maksimalnog pritiska voda. *)
	IF (Rad_PG_KB.Sequence.State = PG_14_Transfer_IEBKB1_BRB2) AND (Rad_PG_KB.Sequence.Substep = 4) THEN
		Rad_PG_KB.Control.PV05.FlushingSP := PGRad.Par.Transfer.PV05StartPressure_bar
			+ ((PGRad.Par.Transfer.PV05FinalPressure_bar - PGRad.Par.Transfer.PV05StartPressure_bar)
			* TIME_TO_REAL(Rad_PG_KB.Timer.Transfer.PV05Guard.ET) / TIME_TO_REAL(Rad_PG_KB.Timer.Transfer.PV05Guard.PT));
	ELSIF (Rad_PG_KB.Sequence.State = PG_01_Priprema_BRB2) AND (Rad_PG_KB.Sequence.Substep = 5) THEN
		Rad_PG_KB.Control.PV05.FlushingSP := PGRad.Par.SetPointPritisakPV05Ispiranje
			+ ((PGRad.Par.SetPointMaxPritisakDolaznaCev - PGRad.Par.SetPointPritisakPV05Ispiranje)
			* TIME_TO_REAL(Rad_PG_KB.Timer.Transfer.PV05Guard.ET) / TIME_TO_REAL(Rad_PG_KB.Timer.Transfer.PV05Guard.PT));
	ELSIF (((Rad_PG_KB.Sequence.State = PG_01_Priprema_BRB2) AND (Rad_PG_KB.Sequence.Substep >= 6))
		OR (Rad_PG_KB.Sequence.State = PG_02_Rad_BRB2)
		OR ((Rad_PG_KB.Sequence.State = PG_03_Zaustavljanje_BRB2) AND NOT PGRad_BRB2.StopSPDostignut)) THEN
		Rad_PG_KB.Control.PV05.FlushingSP := PGRad.Par.SetPointMaxPritisakDolaznaCev;
	ELSIF (Rad_PG_KB.Sequence.BRB2.PreparationState = BRB2_PREP_10_START)
		OR (Rad_PG_KB.Sequence.BRB2.PreparationState = BRB2_PREP_20_ZAGREVANJE)
		OR (Rad_PG_KB.Sequence.BRB2.PreparationState = BRB2_PREP_30_SPReady) THEN
		Rad_PG_KB.Control.PV05.FlushingSP := PGRad.Par.Transfer.PV05StartPressure_bar;
	ELSE
		Rad_PG_KB.Control.PV05.FlushingSP := PGRad.Par.SetPointPritisakPV05Ispiranje;
	END_IF
	Rad_PG_KB.Control.PV05.PID.SetValue := Rad_PG_KB.Control.PV05.FlushingSP; (* Izracunati SP pritiska dolaznog voda. *)
	Rad_PG_KB.Control.PV05.PID();
	IF Rad_PG_KB.Control.PV05.PID.UpdateDone THEN
		Rad_PG_KB.Control.PV05.PID.Update := FALSE;
	END_IF

	(* 8.2) Aktivni ulazni ventil tanka odrzava PT04 po zadrzanom setpoint-u. *)
	Rad_PG_KB.Control.PV_UlazTanka.PID.Enable := ((Rad_PG_KB.Sequence.State = PG_01_Priprema_BRB2) AND (Rad_PG_KB.Sequence.Substep >= 4))
		OR (Rad_PG_KB.Sequence.State = PG_02_Rad_BRB2)
		OR ((Rad_PG_KB.Sequence.State = PG_03_Zaustavljanje_BRB2) AND NOT PGRad_BRB2.StopSPDostignut)
		OR ((Rad_PG_KB.Sequence.State = PG_14_Transfer_IEBKB1_BRB2) AND (Rad_PG_KB.Sequence.Substep = 4));
	Rad_PG_KB.Control.PV_UlazTanka.PID.ActValue := PG.Sens.Pt._4.AI_Output.ScaledValue; (* Merena vrednost PT04. *)
	IF Rad_PG_KB.Sequence.State = PG_14_Transfer_IEBKB1_BRB2 THEN
		Rad_PG_KB.Control.PV_UlazTanka.PID.SetValue := PGRad.Par.Transfer.TankInletPressure_bar;
	ELSE
		Rad_PG_KB.Control.PV_UlazTanka.PID.SetValue := PGRad.Par.SetPointPritisakUlazTanka;
	END_IF;
	Rad_PG_KB.Control.PV_UlazTanka.PID();
	IF Rad_PG_KB.Control.PV_UlazTanka.PID.UpdateDone THEN
		Rad_PG_KB.Control.PV_UlazTanka.PID.Update := FALSE;
	END_IF

	(* 8.3) PID izlazi se upisuju samo kada odgovarajuca sekvenca dozvoljava ventil. *)
	IF Rad_PG_KB.Control.PV05.PID.Enable THEN
		PGRad_Cmd.PropVentili.PV05.SP_Percent := Rad_PG_KB.Control.PV05.PID.Out;
	END_IF
	IF Rad_PG_KB.Control.PV_UlazTanka.PID.Enable THEN
		CASE PGRad.Ctrl.AktivniPropVentilUlazTanka OF
			_01_PG_PV01:
				PGRad_Cmd.Ventili._06_Open := TRUE;
				PGRad_Cmd.PropVentili.PV01.Enable := TRUE;
				PGRad_Cmd.PropVentili.PV01.SP_Percent := Rad_PG_KB.Control.PV_UlazTanka.PID.Out;
			_02_PG_PV02:
				PGRad_Cmd.Ventili._07_Open := TRUE;
				PGRad_Cmd.PropVentili.PV02.Enable := TRUE;
				PGRad_Cmd.PropVentili.PV02.SP_Percent := Rad_PG_KB.Control.PV_UlazTanka.PID.Out;
		END_CASE
	END_IF

	(* -------------------------------------------------------------------------- *)
	(* 9) Adapter RETAIN ulaznih ventila                                         *)
	(* -------------------------------------------------------------------------- *)
	(* Medjusobno iskljucenje V01/V02 stiti od paralelnog spajanja dva izvora. *)
	IF PGRad.CmdRetain.V01_Open AND PGRad.CmdRetain.V02_Open THEN
		PGRad.CmdRetain.V01_Open := FALSE;
		PGRad.CmdRetain.V02_Open := FALSE;
		Rad_PG_KB.Diag.Fault.Latched := TRUE;
		Rad_PG_KB.Diag.Fault.Code := 10;
		Rad_PG_KB.Diag.Fault.Text := 'PG_V01 i PG_V02 istovremeno zahtevani';
	END_IF;

	(* -------------------------------------------------------------------------- *)
	(* 10) Fault/reset politika                                                   *)
	(* -------------------------------------------------------------------------- *)
	(* Rad_PG_KB.HMI.Cntrl.Reset se prosledjuje AirRelease blokovima preko ResetAll. Procesni  *)
	(* Rad_PG_KB.Diag.Fault.Latched u pregledanom kodu nema implementirano brisanje/reset.        *)

	(* -------------------------------------------------------------------------- *)
	(* 11) Procesni status za Communication/HMI task                             *)
	(* -------------------------------------------------------------------------- *)
	(* Enum Rad_PG_KB.Sequence.State se preslikava u stabilan brojcani status AsIMA/HMI ugovora. *)
	CASE Rad_PG_KB.Sequence.State OF
		PG_01_Priprema_BRB2:
			PGRad_Status.State := 1;
			PGRad_Status.StateComment := 'STANJE: PRIPREMA BRB2';
		PG_02_Rad_BRB2:
			PGRad_Status.State := 2;
			PGRad_Status.StateComment := 'STANJE: RAD BRB2';
		PG_03_Zaustavljanje_BRB2:
			PGRad_Status.State := 3;
			PGRad_Status.StateComment := 'STANJE: ZAUSTAVLJANJE BRB2';
		PG_11_Priprema_IEBKB1:
			PGRad_Status.State := 11;
			PGRad_Status.StateComment := 'STANJE: PRIPREMA IEBKB1';
		PG_12_Rad_IEBKB1:
			PGRad_Status.State := 12;
			PGRad_Status.StateComment := 'STANJE: RAD IEBKB1';
		PG_13_Zaustavljanje_IEBKB1:
			PGRad_Status.State := 13;
			PGRad_Status.StateComment := 'STANJE: ZAUSTAVLJANJE IEBKB1';
		PG_14_Transfer_IEBKB1_BRB2:
			PGRad_Status.State := 14;
			PGRad_Status.StateComment := 'STANJE: TRANSFER IEBKB1 NA BRB2';
	ELSE
		PGRad_Status.State := 0;
		PGRad_Status.StateComment := 'STANJE: STANDBY';
	END_CASE
	PGRad_Status.Substep := Rad_PG_KB.Sequence.Substep;

	CASE Rad_PG_KB.Sequence.State OF
		PG_00_Stand_By:
			PGRad_Status.SubstepComment := 'PODKORAK: Ceka komandu START';

		PG_01_Priprema_BRB2:
			CASE Rad_PG_KB.Sequence.Substep OF
				0: PGRad_Status.SubstepComment := 'PODKORAK: Ulazak u pripremu BRB2';
				1: PGRad_Status.SubstepComment := 'PODKORAK: Ceka zatvaranje PG_V01';
				2: PGRad_Status.SubstepComment := 'PODKORAK: Ceka otvaranje PG_V02';
				3: PGRad_Status.SubstepComment := 'PODKORAK: Ispiranje BRB2 grane';
				4: PGRad_Status.SubstepComment := 'PODKORAK: Priprema ulaza prihvatnog tanka';
				5: PGRad_Status.SubstepComment := 'PODKORAK: Mek prelaz pritiska PG_PV05';
				6: PGRad_Status.SubstepComment := 'PODKORAK: Punjenje prihvatnog tanka';
			ELSE
				PGRad_Status.SubstepComment := 'PODKORAK: Nepoznata priprema BRB2';
			END_CASE

		PG_14_Transfer_IEBKB1_BRB2:
			PGRad_Status.SubstepComment := 'PODKORAK: Transfer IEBKB1 na BRB2';

		PG_02_Rad_BRB2:
			IF Rad_PG_KB.Sequence.Substep = 0 THEN
				PGRad_Status.SubstepComment := 'PODKORAK: Pokretanje izlazne pumpe';
			ELSE
				PGRad_Status.SubstepComment := 'PODKORAK: Regulacija i odrzavanje rada';
			END_IF

		PG_03_Zaustavljanje_BRB2:
			PGRad_Status.SubstepComment := 'PODKORAK: Kontrolisano zaustavljanje BRB2';

		PG_11_Priprema_IEBKB1:
			CASE Rad_PG_KB.Sequence.Substep OF
				0: PGRad_Status.SubstepComment := 'PODKORAK: Ulazak u pripremu IEBKB1';
				1: PGRad_Status.SubstepComment := 'PODKORAK: Ceka zatvaranje PG_V02';
				2: PGRad_Status.SubstepComment := 'PODKORAK: Ceka otvaranje PG_V01';
				3: PGRad_Status.SubstepComment := 'PODKORAK: Ceka pocetak dotoka IEBKB1';
				4: PGRad_Status.SubstepComment := 'PODKORAK: Punjenje prihvatnog tanka';
			ELSE
				PGRad_Status.SubstepComment := 'PODKORAK: Nepoznata priprema IEBKB1';
			END_CASE

		PG_12_Rad_IEBKB1:
			IF Rad_PG_KB.Sequence.Substep = 0 THEN
				PGRad_Status.SubstepComment := 'PODKORAK: Pokretanje izlazne pumpe';
			ELSE
				PGRad_Status.SubstepComment := 'PODKORAK: Regulacija i odrzavanje rada';
			END_IF

		PG_13_Zaustavljanje_IEBKB1:
			CASE Rad_PG_KB.Sequence.Substep OF
				0: PGRad_Status.SubstepComment := 'PODKORAK: Ulazak u zaustavljanje IEBKB1';
				1: PGRad_Status.SubstepComment := 'PODKORAK: Ceka prestanak dotoka IEBKB1';
				2: PGRad_Status.SubstepComment := 'PODKORAK: Ceka zatvaranje PG_V05';
				3: PGRad_Status.SubstepComment := 'PODKORAK: Ceka zatvaranje PG_V01';
			ELSE
				PGRad_Status.SubstepComment := 'PODKORAK: Nepoznat stop IEBKB1';
			END_CASE

	ELSE
		PGRad_Status.SubstepComment := 'PODKORAK: Nepoznato stanje sistema';
	END_CASE
	PGRad_Status.Fault := Rad_PG_KB.Diag.Fault.Latched;
	PGRad_Status.FaultCode := Rad_PG_KB.Diag.Fault.Code;
	CASE Rad_PG_KB.Sequence.BRB2.PreparationState OF
		BRB2_PREP_10_START:
			PGRad_Status.BRB2PreparationState := 10;
			PGRad_Status.BRB2PreparationStateComment := 'BRB2 PRIPREMA: START I CEKANJE PROTOKA';
		BRB2_PREP_20_ZAGREVANJE:
			PGRad_Status.BRB2PreparationState := 20;
			PGRad_Status.BRB2PreparationStateComment := 'BRB2 PRIPREMA: ZAGREVANJE CEVOVODA';
		BRB2_PREP_30_SPReady:
			PGRad_Status.BRB2PreparationState := 30;
			PGRad_Status.BRB2PreparationStateComment := 'BRB2 PRIPREMA: SP SPREMAN ZA TRANSFER';
		BRB2_PREP_40_STOPPING:
			PGRad_Status.BRB2PreparationState := 40;
			PGRad_Status.BRB2PreparationStateComment := 'BRB2 PRIPREMA: KONTROLISANO ZAUSTAVLJANJE';
		BRB2_PREP_90_FAULT:
			PGRad_Status.BRB2PreparationState := 90;
			PGRad_Status.BRB2PreparationStateComment := 'BRB2 PRIPREMA: FAULT';
	ELSE
		PGRad_Status.BRB2PreparationState := 0;
		PGRad_Status.BRB2PreparationStateComment := 'BRB2 PRIPREMA: IDLE';
	END_CASE
	PGRad_Status.BRB2Ready := Rad_PG_KB.Sequence.BRB2.Ready;
	PGRad_Status.IEBKB1InterfaceReady := PGRad_IEBKB1Prepared.Enable
		AND PGRad_IEBKB1Prepared.InterfaceReady
		AND PGRad_IEBKB1Prepared.CommValid
		AND PGRad_IEBKB1Prepared.HeartbeatValid
		AND NOT PGRad_IEBKB1Prepared.Fault;
	PGRad_Status.TransferBlocked := Rad_PG_KB.Sequence.BRB2.Ready AND NOT PGRad_Status.IEBKB1InterfaceReady;

END_PROGRAM
```

#### Variables.var - Local variables
```iecst
VAR
	(* Jedina lokalna instanca: svi HMI, sekvencni, regulacioni, statusni, dijagnosticki i vremenski podaci programa. *)
	Rad_PG_KB : typRadPGKB;
	BootInfoFB : SysInfo; (* Jednokratno citanje uzroka restarta u Init.st za AutoRestart (INIT_REASON_WARMSTART). *)
END_VAR
```

#### Init.st
```iecst
PROGRAM _INIT
	(* ======================================================================== *)
	(* 1) Inicijalizacija izvrsnog konteksta                                     *)
	(* ======================================================================== *)
	Rad_PG_KB.Sequence.State := PG_00_Stand_By;
	Rad_PG_KB.Sequence.Substep := 0;

	Rad_PG_KB.HMI.Cntrl.Start := FALSE;
	Rad_PG_KB.HMI.Cntrl.Stop := FALSE;
	Rad_PG_KB.HMI.Cntrl.Reset := FALSE;
	Rad_PG_KB.HMI.Cntrl.SetDefaultParameters := FALSE;
	Rad_PG_KB.HMI.Cntrl.PrepareBRB2 := FALSE;
	Rad_PG_KB.HMI.Cntrl.TransferToBRB2 := FALSE;
	Rad_PG_KB.HMI.Cntrl.Continue := FALSE;
	Rad_PG_KB.Sequence.BRB2.PreparationState := BRB2_PREP_00_IDLE;
	Rad_PG_KB.Sequence.BRB2.PreparationSubstep := 0;
	Rad_PG_KB.Sequence.BRB2.Ready := FALSE;
	Rad_PG_KB.Sequence.Transfer.Requested := FALSE;
	IF PGRad.Ctrl.BRB2Regulacija = BRB2_00_NEAKTIVNA THEN
		PGRad.Ctrl.BRB2Regulacija := BRB2_01_REG_PROTOK;
	END_IF;
	IF PGRad.Ctrl.SelektovaniIzvor = _02_IEBKB1 THEN
		Rad_PG_KB.HMI.Cntrl.SelectIEBKB1 := TRUE;
	ELSE
		Rad_PG_KB.HMI.Cntrl.SelectIEBKB1 := FALSE;
		PGRad.Ctrl.SelektovaniIzvor := _01_BRB2;
	END_IF;

	(* -------------------------------------------------------------------------- *)
	(* 2) Detekcija uzroka restarta za automatski start (PGRad.Ctrl.AutoRestart)  *)
	(* -------------------------------------------------------------------------- *)
	(* WARMSTART = restart posle nestanka struje; ne okida se na cold start/download. *)
	BootInfoFB(enable := TRUE);
	Rad_PG_KB.AutoRestart.WarmstartDetected := (BootInfoFB.init_reason = INIT_REASON_WARMSTART);
	Rad_PG_KB.AutoRestart.Timer.IN := FALSE;

	Rad_PG_KB.Diag.Fault.Latched := FALSE;
	Rad_PG_KB.Diag.Fault.Code := 0;
	Rad_PG_KB.Diag.Fault.Text := '';
	Rad_PG_KB.Timer.PG_V01.Close(IN := FALSE, PT := T#0s);
	Rad_PG_KB.Timer.PG_V02.Open(IN := FALSE, PT := T#0s);
	Rad_PG_KB.Timer.Transfer.PV05Guard(IN := FALSE, PT := T#0s);
	Rad_PG_KB.Timer.BRB2.PreparationFlow(IN := FALSE, PT := T#0s);
	Rad_PG_KB.Timer.BRB2.TemperatureAlarm(IN := FALSE, PT := T#0s);
	Rad_PG_KB.Timer.BRB2.TemperatureStop(IN := FALSE, PT := T#0s);
	Rad_PG_KB.Timer.BRB2.PressureAlarm(IN := FALSE, PT := T#0s);
	Rad_PG_KB.Timer.BRB2.PressureStop(IN := FALSE, PT := T#0s);
	Rad_PG_KB.Timer.Transfer.Flow(IN := FALSE, PT := T#0s);
	Rad_PG_KB.Control.PV05.FlushingSP := 0.0;
	Rad_PG_KB.Status.PV05.FlushingOpened := FALSE;
	Rad_PG_KB.Status.Pump.OutletStopped := FALSE;

	(* ======================================================================== *)
	(* 2) Inicijalizacija PID parametara proporcionalnih ventila                *)
	(* ======================================================================== *)
	(* PV05 cuva pritisak dolaznog voda, a aktivni ulazni PV odrzava PT04. *)
	(* FilterTime filtrira D clan i nema uticaja dok je DerivativeTime = 0.0. *)
	Rad_PG_KB.Control.PV05.PID.MinOut := 0.0;
	Rad_PG_KB.Control.PV05.PID.MaxOut := 100.0;
	Rad_PG_KB.Control.PV05.PID.PIDParameters.DerivativeTime := 0.0;
	Rad_PG_KB.Control.PV05.PID.PIDParameters.FilterTime := 10.0;
	Rad_PG_KB.Control.PV05.PID.PIDParameters.Gain := 1.0;
	Rad_PG_KB.Control.PV05.PID.PIDParameters.IntegrationTime := 180.0;
	Rad_PG_KB.Control.PV05.PID.Invert := TRUE;
	Rad_PG_KB.Control.PV05.PID.Update := TRUE;

	Rad_PG_KB.Control.PV_UlazTanka.PID.MinOut := 0.0;
	Rad_PG_KB.Control.PV_UlazTanka.PID.MaxOut := 100.0;
	Rad_PG_KB.Control.PV_UlazTanka.PID.PIDParameters.DerivativeTime := 0.0;
	Rad_PG_KB.Control.PV_UlazTanka.PID.PIDParameters.FilterTime := 10.0;
	Rad_PG_KB.Control.PV_UlazTanka.PID.PIDParameters.Gain := 1.0;
	Rad_PG_KB.Control.PV_UlazTanka.PID.PIDParameters.IntegrationTime := 180.0;
	Rad_PG_KB.Control.PV_UlazTanka.PID.Invert := FALSE;
	Rad_PG_KB.Control.PV_UlazTanka.PID.Update := TRUE;

	(* ======================================================================== *)
	(* 3) Obnova RETAIN komandi bistabilnih ulaznih ventila                      *)
	(* ======================================================================== *)
	(* RETAIN polozaji se neposredno prenose na bistabilne ulazne ventile. *)
	PG.Act.AV._1.Open := PGRad.CmdRetain.V01_Open; (* PG_V01: dolaz sa IEBKB1. *)
	PG.Act.AV._2.Open := PGRad.CmdRetain.V02_Open; (* PG_V02: dolaz sa BRB2. *)

	(* ======================================================================== *)
	(* 4) Bezbedan reset neretentivnog upravljackog vektora                      *)
	(* ======================================================================== *)
	PGRad_Cmd.Aktivan := FALSE;
	PGRad_Cmd.Ventili._03_Open := FALSE;
	PGRad_Cmd.Ventili._04_Open := FALSE;
	PGRad_Cmd.Ventili._05_Open := FALSE;
	PGRad_Cmd.Ventili._06_Open := FALSE;
	PGRad_Cmd.Ventili._07_Open := FALSE;

	PGRad_Cmd.PropVentili.PV01.Enable := FALSE;
	PGRad_Cmd.PropVentili.PV02.Enable := FALSE;
	PGRad_Cmd.PropVentili.PV05.Enable := FALSE;
	PGRad_Cmd.AirRelease.PV03.Enable := FALSE;
	PGRad_Cmd.AirRelease.PV04.Enable := FALSE;
	PGRad_Cmd.AirRelease.UseIEBKB1Parameters := FALSE;
	PGRad_Cmd.AirRelease.ResetAll := FALSE;

	PGRad_Cmd.Pumpe._01.Run := FALSE;
	PGRad_Cmd.Pumpe._02.Run := FALSE;
	PGRad_Cmd.PID.Enable := FALSE;
	PGRad_Cmd.PID.ActValue := 0.0;
	PGRad_Cmd.PID.SetValue := 0.0;
	PGRad_Cmd.PID.Invert := FALSE;
	PGRad_Cmd.PID.MaxOut := 0.0;
	PGRad_Cmd.PID.EnableTracking := FALSE;
	PGRad_Cmd.PID.TrackingValue := 0.0;
	PGRad_BRB2Cmd.ZahtevZaustavljanja := FALSE;
	PGRad_BRB2Cmd.VentiliPodstaniceZatvoreni := FALSE;

	(* ======================================================================== *)
	(* 5) Cold-boot provera RETAIN parametara                                   *)
	(* ======================================================================== *)
	(* RETAIN parametri se inicijalizuju i na cold boot-u. *)
	IF (PGRad.Par.SetPritisakPotisa <= 0.0)
		OR (PGRad.Par.MaxFR_Pumpe <= 0.0)
		OR (PGRad.Par.SetPointPritisakPV05Ispiranje <= 0.0)
		OR (PGRad.Par.SetPointPritisakUlazTanka <= 0.0)
		OR (PGRad.Par.SetPointNivoTankaUpozorenje <= 0.0)
		OR (PGRad.Par.BRB2Preparation.MinTemperature_degC <= 0.0)
		OR (PGRad.Par.BRB2Preparation.FlowTimeout_s <= 0.0)
		OR (PGRad.Par.Transfer.PV05StartPressure_bar <= 0.0)
		OR (PGRad.Par.Transfer.PV05FinalPressure_bar <= 0.0)
		OR (PGRad.Par.Transfer.TankInletPressure_bar <= 0.0)
		OR (PGRad.Par.Transfer.PressureRamp_s <= 0.0)
		OR (PGRad.Par.TimeSP.PrelazPV05Cuvar_s <= 0.0)
		OR (PGRad.Par.PocetnaFrekvencaIzlaznePumpe <= 0.0)
		OR (PGRad.Par.MaxOtvorPropZaZatvaranje <= 0.0)
		OR (PGRad.Par.TimeSP.OverlapPumpi_s <= 0.0)
		OR (PGRad.Par.TimeSP.AutoRestartDelay_s <= 0.0)
		OR (PGRad.Par.TimeSP.ValvePositionTimeout_s <= 0.0)
		OR (PGRad.Par.TimeSP.InterlockDebounce_s <= 0.0)
		OR (PGRad.Par.AirRelease.BRB2.PV03.NumberOfLS = 0)
		OR (PGRad.Par.AirRelease.BRB2.PV04.NumberOfLS = 0)
		OR (PGRad.Par.AirRelease.IEBKB1.PV03.NumberOfLS = 0)
		OR (PGRad.Par.AirRelease.IEBKB1.PV04.NumberOfLS = 0) THEN
		Rad_PG_KB.HMI.Cntrl.SetDefaultParameters := TRUE;
	END_IF

END_PROGRAM
```

#### Exit.st
```iecst
PROGRAM _EXIT
	(* Nema zavrsne akcije: bezbedne komande se postavljaju u svakom cyclic scan-u. *)
END_PROGRAM
```

### Program Logical/Project/PG_Intf (IEC)

#### Cyclic.st
```iecst
PROGRAM _CYCLIC
	(* ======================================================================== *)
	(* PG_INTF - PT/BRB2 KOMUNIKACIONI UGOVOR                                 *)
	(* COMMON: lokalni PGRad ugovor i brojači snapshot-a.                     *)
	(* MANUAL: prenosi ManualMode, Start, Stop, NextStep i Abort ka BRB2.      *)
	(* AUTO: prenosi procesne zahteve, regulacioni PV/SP i izbor izvora.       *)
	(* STOP/FAULT: watchdog status BRB2 se koristi kao komunikacioni fault.    *)
	(* STATUS: Rx statusi se prihvataju samo dok je udaljeni watchdog validan.  *)
	(* ======================================================================== *)
	(* ======================================================================== *)
	(* 1) Lokalni PT-BRB2 procesni ugovor                                       *)
	(* ======================================================================== *)
	(* PGRad_BRB2Cmd je jedini lokalni izvor komandi. Ovaj program preslikava   *)
	(* komande u zajednicki procesni prikaz koji koristi master sekvenca.       *)
	PGRad_BRB2.RadKaPodstanici := PGRad_BRB2Cmd.RadKaPodstanici;
	PGRad_BRB2.ManualMode := PGRad_BRB2Cmd.ManualMode;
	PGRad_BRB2.ManualSequence := PGRad_BRB2Cmd.ManualSequence;
	PGRad_BRB2.ManualStart := PGRad_BRB2Cmd.ManualStart;
	PGRad_BRB2.ManualStop := PGRad_BRB2Cmd.ManualStop;
	PGRad_BRB2.ManualNextStep := PGRad_BRB2Cmd.ManualNextStep;
	PGRad_BRB2.ManualAbort := PGRad_BRB2Cmd.ManualAbort;
	PGRad_BRB2.ZahtevStarta := PGRad_BRB2Cmd.ZahtevStarta;
	PGRad_BRB2.ZahtevZaustavljanja := PGRad_BRB2Cmd.ZahtevZaustavljanja;
	PGRad_BRB2.VentiliPodstaniceZatvoreni := PGRad_BRB2Cmd.VentiliPodstaniceZatvoreni;
	PGRad_BRB2.PritisakIEBKB1 := PGRad_BRB2Cmd.PritisakIEBKB1;
	PGRad_BRB2.PodstanicaURezimuRada := PGRad_BRB2Cmd.PodstanicaURezimuRada;
	CASE PGRad_BRB2Cmd.RegulationMode OF
		BRB2_01_REG_PROTOK: PGRad_BRB2.RegulationMode := 1;
		BRB2_02_REG_NIVO: PGRad_BRB2.RegulationMode := 2;
		BRB2_03_REG_TEMPERATURA: PGRad_BRB2.RegulationMode := 3;
		ELSE PGRad_BRB2.RegulationMode := 0;
	END_CASE;
	PGRad_BRB2.RegulationPV := PGRad_BRB2Cmd.RegulationPV;
	PGRad_BRB2.RegulationSP := PGRad_BRB2Cmd.RegulationSP;
	PGRad_BRB2.RegulationPVValid := PGRad_BRB2Cmd.RegulationPVValid;
	PGRad_BRB2.RegulationInvert := PGRad_BRB2Cmd.RegulationInvert;
	PGRad_BRB2.NivoPrihvatniSud := PGRad_BRB2Cmd.NivoPrihvatniSud;
	(* Brojac se menja svakim ciklusom i udaljenom PLC-u dokazuje da snapshot   *)
	(* nije samo poslednja zadrzana vrednost nakon prekida komunikacije.        *)
	PGRad_BRB2Cmd.CommandCounter := PGRad_BRB2Cmd.CommandCounter + 1;
	PGRad_BRB2.CommandCounter := PGRad_BRB2Cmd.CommandCounter;

	(* ======================================================================== *)
	(* 2) PT izlazni AsIMA snapshot                                             *)
	(* ======================================================================== *)
	(* Tx struktura je jedini komunikacioni izlaz Podstanice prema BRB2.        *)
	(* Odvajanje od lokalnog prikaza sprecava vise pisaca nad istim podacima.   *)
	PGRad_BRB2_Tx.RadKaPodstanici := PGRad_BRB2Cmd.RadKaPodstanici;
	PGRad_BRB2_Tx.ManualMode := PGRad_BRB2Cmd.ManualMode;
	PGRad_BRB2_Tx.ManualSequence := PGRad_BRB2Cmd.ManualSequence;
	PGRad_BRB2_Tx.ManualStart := PGRad_BRB2Cmd.ManualStart;
	PGRad_BRB2_Tx.ManualStop := PGRad_BRB2Cmd.ManualStop;
	PGRad_BRB2_Tx.ManualNextStep := PGRad_BRB2Cmd.ManualNextStep;
	PGRad_BRB2_Tx.ManualAbort := PGRad_BRB2Cmd.ManualAbort;
	PGRad_BRB2_Tx.CommandCounter := PGRad_BRB2Cmd.CommandCounter;
	PGRad_BRB2_Tx.ZahtevStarta := PGRad_BRB2Cmd.ZahtevStarta;
	PGRad_BRB2_Tx.ZahtevZaustavljanja := PGRad_BRB2Cmd.ZahtevZaustavljanja;
	PGRad_BRB2_Tx.VentiliPodstaniceZatvoreni := PGRad_BRB2Cmd.VentiliPodstaniceZatvoreni;
	PGRad_BRB2_Tx.PritisakIEBKB1 := PGRad_BRB2Cmd.PritisakIEBKB1;
	PGRad_BRB2_Tx.PodstanicaURezimuRada := PGRad_BRB2Cmd.PodstanicaURezimuRada;
	CASE PGRad_BRB2Cmd.RegulationMode OF
		BRB2_01_REG_PROTOK: PGRad_BRB2_Tx.RegulationMode := 1;
		BRB2_02_REG_NIVO: PGRad_BRB2_Tx.RegulationMode := 2;
		BRB2_03_REG_TEMPERATURA: PGRad_BRB2_Tx.RegulationMode := 3;
		ELSE PGRad_BRB2_Tx.RegulationMode := 0;
	END_CASE;
	PGRad_BRB2_Tx.RegulationPV := PGRad_BRB2Cmd.RegulationPV;
	PGRad_BRB2_Tx.RegulationSP := PGRad_BRB2Cmd.RegulationSP;
	PGRad_BRB2_Tx.RegulationPVValid := PGRad_BRB2Cmd.RegulationPVValid;
	PGRad_BRB2_Tx.RegulationInvert := PGRad_BRB2Cmd.RegulationInvert;
	PGRad_BRB2_Tx.NivoPrihvatniSud := PGRad_BRB2Cmd.NivoPrihvatniSud;

	(* ======================================================================== *)
	(* 3) BRB2 ulazni procesni status                                           *)
	(* ======================================================================== *)
	(* 3.1) StatusCounter mora da se menja; zadrzan snapshot duze od 5 s nije validna veza. *)
	(* Svaka promena ponovo pokrece vremenski nadzor. Nepromenjen brojac drzi    *)
	(* TON aktivnim sve dok se ne potvrdi timeout komunikacionog statusa.       *)
	IF PGRad_BRB2_Rx.StatusCounter <> PGRad_BRB2Watchdog.LastCounter THEN
		PGRad_BRB2Watchdog.LastCounter := PGRad_BRB2_Rx.StatusCounter;
		PGRad_BRB2Watchdog.ReceivedOnce := TRUE;
		PGRad_BRB2Watchdog.ReceiveTimeout.IN := FALSE;
	ELSE
		PGRad_BRB2Watchdog.ReceiveTimeout.IN := TRUE;
	END_IF;
	PGRad_BRB2Watchdog.ReceiveTimeout.PT := T#5s;
	PGRad_BRB2Watchdog.ReceiveTimeout();
	PGRad_BRB2Watchdog.Valid :=
		PGRad_BRB2Watchdog.ReceivedOnce AND NOT PGRad_BRB2Watchdog.ReceiveTimeout.Q;

	(* 3.2) Lokalni proces prihvata BRB2 status samo dok je komunikacija validna. *)
	IF PGRad_BRB2Watchdog.Valid THEN
		PGRad_BRB2.PumpaAktivna := PGRad_BRB2_Rx.PumpaAktivna;
		PGRad_BRB2.IspiranjeProtokDostignut := PGRad_BRB2_Rx.IspiranjeProtokDostignut;
		PGRad_BRB2.IspiranjeMinTrajanjeDostignuto := PGRad_BRB2_Rx.IspiranjeMinTrajanjeDostignuto;
		PGRad_BRB2.StopSPDostignut := PGRad_BRB2_Rx.StopSPDostignut;
		PGRad_BRB2.RB2V01Zatvoren := PGRad_BRB2_Rx.RB2V01Zatvoren;
		PGRad_BRB2.RB2V02Zatvoren := PGRad_BRB2_Rx.RB2V02Zatvoren;
		PGRad_BRB2.StatusCounter := PGRad_BRB2_Rx.StatusCounter;
		PGRad_BRB2.BRB2Fault := PGRad_BRB2_Rx.BRB2Fault;
		PGRad_BRB2.BRB2FaultCode := PGRad_BRB2_Rx.BRB2FaultCode;
		PGRad_BRB2.RegulationPVFault := PGRad_BRB2_Rx.RegulationPVFault;
	ELSE
		PGRad_BRB2.PumpaAktivna := FALSE;
		PGRad_BRB2.IspiranjeProtokDostignut := FALSE;
		PGRad_BRB2.IspiranjeMinTrajanjeDostignuto := FALSE;
		PGRad_BRB2.StopSPDostignut := FALSE;
		PGRad_BRB2.RB2V01Zatvoren := FALSE;
		PGRad_BRB2.RB2V02Zatvoren := FALSE;
		PGRad_BRB2.StatusCounter := 0;
		PGRad_BRB2.BRB2Fault := TRUE;
		PGRad_BRB2.BRB2FaultCode := 3; (* Gubitak komunikacije sa BRB2. *)
		PGRad_BRB2.RegulationPVFault := FALSE;
	END_IF;
END_PROGRAM
```

#### Init.st
```iecst
PROGRAM _INIT
	(* Inicijalizacija BRB2 watchdog-a; status je nevalidan do prve promene udaljenog brojača. *)
	PGRad_BRB2Watchdog.LastCounter := 0;
	PGRad_BRB2Watchdog.ReceivedOnce := FALSE;
	PGRad_BRB2Watchdog.ReceiveTimeout(IN := FALSE, PT := T#5s);
	PGRad_BRB2Watchdog.Valid := FALSE;
END_PROGRAM
```

### Program Logical/Project/HMI_Svc (IEC)

#### Init.st - Init code
```iecst
PROGRAM _INIT
	(* ======================================================================== *)
	(* 1) Inicijalizacija Podstanica trend prikaza                              *)
	(* ======================================================================== *)
	PGRad_TrendCursor.Position := 0.5;
	PGRad_TrendCursor.ViewSpan := 14400;
	PGRad_TrendCursor.PreviousViewSpan := 14400;
	PGRad_TrendCursor.FollowNow := TRUE;
	PGRad_TrendCursor.CmdBack := FALSE;
	PGRad_TrendCursor.CmdForward := FALSE;
	PGRad_TrendCursor.CmdNow := FALSE;
	AlarmCmdAcknowledge := FALSE;
	AlarmCmdResetRecords := FALSE;
	AlarmCmdResetDevices := FALSE;
	AlarmCmdResetProcess := FALSE;
END_PROGRAM
```

#### Cyclic.st - Cyclic code
```iecst
PROGRAM _CYCLIC
	(* ======================================================================== *)
	(* 1) Rezim i raspolozivi vremenski opseg Podstanica trenda                 *)
	(* ======================================================================== *)
	(* VC pri otvaranju continuous trenda postavlja mod 1; mod 0 drzi zadati prozor. *)
	PGRad_TrendCursor.AxisMode := 0;

	TrendClock.enable := TRUE;
	TrendClock();
	TrendNow_s := DT_TO_UDINT(TrendClock.DT1);
	IF TrendNow_s > 864000 THEN
		TrendEarliest_s := TrendNow_s - 864000;
	ELSE
		TrendEarliest_s := 0;
	END_IF;
	IF (DT_TO_UDINT(PGRad_TrendCursor.RecordingStart) > TrendEarliest_s)
		AND (DT_TO_UDINT(PGRad_TrendCursor.RecordingStart) <= TrendNow_s) THEN
		TrendEarliest_s := DT_TO_UDINT(PGRad_TrendCursor.RecordingStart);
	END_IF;

	(* ======================================================================== *)
	(* 2) Zoom i navigacija vremenskog prozora                                  *)
	(* ======================================================================== *)
	IF PGRad_TrendCursor.ViewSpan < 3600 THEN
		PGRad_TrendCursor.ViewSpan := 3600;
	ELSIF PGRad_TrendCursor.ViewSpan > 172800 THEN
		PGRad_TrendCursor.ViewSpan := 172800;
	END_IF;

	IF (DT_TO_UDINT(PGRad_TrendCursor.ViewStart) = 0)
		AND (TrendNow_s >= DINT_TO_UDINT(PGRad_TrendCursor.ViewSpan)) THEN
		PGRad_TrendCursor.ViewStart := UDINT_TO_DT(
			TrendNow_s - DINT_TO_UDINT(PGRad_TrendCursor.ViewSpan));
		PGRad_TrendCursor.FollowNow := FALSE;
	END_IF;

	IF PGRad_TrendCursor.ViewSpan <> PGRad_TrendCursor.PreviousViewSpan THEN
		IF PGRad_TrendCursor.FollowNow THEN
			PGRad_TrendCursor.ViewStart := UDINT_TO_DT(
				TrendNow_s - DINT_TO_UDINT(PGRad_TrendCursor.ViewSpan));
		ELSE
			PGRad_TrendCursor.ViewStart := UDINT_TO_DT(
				DT_TO_UDINT(PGRad_TrendCursor.ViewStart)
				+ DINT_TO_UDINT(PGRad_TrendCursor.PreviousViewSpan)
				- DINT_TO_UDINT(PGRad_TrendCursor.ViewSpan));
		END_IF;
		PGRad_TrendCursor.PreviousViewSpan := PGRad_TrendCursor.ViewSpan;
		PGRad_TrendCursor.FollowNow := FALSE;
	END_IF;

	IF PGRad_TrendCursor.CmdNow THEN
		IF TrendNow_s >= DINT_TO_UDINT(PGRad_TrendCursor.ViewSpan) THEN
			PGRad_TrendCursor.ViewStart := UDINT_TO_DT(
				TrendNow_s - DINT_TO_UDINT(PGRad_TrendCursor.ViewSpan));
		END_IF;
		PGRad_TrendCursor.FollowNow := FALSE;
	END_IF;

	IF PGRad_TrendCursor.CmdBack THEN
		PGRad_TrendCursor.FollowNow := FALSE;
		IF DT_TO_UDINT(PGRad_TrendCursor.ViewStart) > (TrendEarliest_s + DINT_TO_UDINT(PGRad_TrendCursor.ViewSpan)) THEN
			PGRad_TrendCursor.ViewStart := UDINT_TO_DT(
				DT_TO_UDINT(PGRad_TrendCursor.ViewStart) - DINT_TO_UDINT(PGRad_TrendCursor.ViewSpan));
		ELSE
			PGRad_TrendCursor.ViewStart := UDINT_TO_DT(TrendEarliest_s);
		END_IF;
	END_IF;

	IF PGRad_TrendCursor.CmdForward THEN
		IF (DT_TO_UDINT(PGRad_TrendCursor.ViewStart) + (2 * DINT_TO_UDINT(PGRad_TrendCursor.ViewSpan))) >= TrendNow_s THEN
			PGRad_TrendCursor.ViewStart := UDINT_TO_DT(
				TrendNow_s - DINT_TO_UDINT(PGRad_TrendCursor.ViewSpan));
			PGRad_TrendCursor.FollowNow := FALSE;
		ELSE
			PGRad_TrendCursor.ViewStart := UDINT_TO_DT(
				DT_TO_UDINT(PGRad_TrendCursor.ViewStart) + DINT_TO_UDINT(PGRad_TrendCursor.ViewSpan));
		END_IF;
	END_IF;

	(* ======================================================================== *)
	(* 3) Oznake vremenske ose i apsolutno vreme kursora                        *)
	(* ======================================================================== *)
	PGRad_TrendCursor.AxisTime0 := PGRad_TrendCursor.ViewStart;
	PGRad_TrendCursor.AxisTime1 := UDINT_TO_DT(
		DT_TO_UDINT(PGRad_TrendCursor.ViewStart) + (DINT_TO_UDINT(PGRad_TrendCursor.ViewSpan) / 8));
	PGRad_TrendCursor.AxisTime2 := UDINT_TO_DT(
		DT_TO_UDINT(PGRad_TrendCursor.ViewStart) + ((2 * DINT_TO_UDINT(PGRad_TrendCursor.ViewSpan)) / 8));
	PGRad_TrendCursor.AxisTime3 := UDINT_TO_DT(
		DT_TO_UDINT(PGRad_TrendCursor.ViewStart) + ((3 * DINT_TO_UDINT(PGRad_TrendCursor.ViewSpan)) / 8));
	PGRad_TrendCursor.AxisTime4 := UDINT_TO_DT(
		DT_TO_UDINT(PGRad_TrendCursor.ViewStart) + ((4 * DINT_TO_UDINT(PGRad_TrendCursor.ViewSpan)) / 8));
	PGRad_TrendCursor.AxisTime5 := UDINT_TO_DT(
		DT_TO_UDINT(PGRad_TrendCursor.ViewStart) + ((5 * DINT_TO_UDINT(PGRad_TrendCursor.ViewSpan)) / 8));
	PGRad_TrendCursor.AxisTime6 := UDINT_TO_DT(
		DT_TO_UDINT(PGRad_TrendCursor.ViewStart) + ((6 * DINT_TO_UDINT(PGRad_TrendCursor.ViewSpan)) / 8));
	PGRad_TrendCursor.AxisTime7 := UDINT_TO_DT(
		DT_TO_UDINT(PGRad_TrendCursor.ViewStart) + ((7 * DINT_TO_UDINT(PGRad_TrendCursor.ViewSpan)) / 8));
	PGRad_TrendCursor.AxisTime8 := UDINT_TO_DT(
		DT_TO_UDINT(PGRad_TrendCursor.ViewStart) + DINT_TO_UDINT(PGRad_TrendCursor.ViewSpan));

	(* VC vraca vreme kursora u ms od pocetka referentnog trend zapisa. *)
	PGRad_TrendCursor.DateTime := UDINT_TO_DT(
		DT_TO_UDINT(PGRad_TrendCursor.RecordingStart)
		+ (PGRad_TrendCursor.Time / 1000));

	PGRad_TrendCursor.CmdBack := FALSE;
	PGRad_TrendCursor.CmdForward := FALSE;
	PGRad_TrendCursor.CmdNow := FALSE;

	(* ======================================================================== *)
	(* 4) Alarmne komande i status za VC                                        *)
	(* ======================================================================== *)
	IF AlarmCmdAcknowledge THEN
		PT_Alarm.Cmd.AcknowledgeAll := TRUE;
		AlarmCmdAcknowledge := FALSE;
	END_IF;
	IF AlarmCmdResetRecords THEN
		PT_Alarm.Cmd.ResetAlarmRecords := TRUE;
		AlarmCmdResetRecords := FALSE;
	END_IF;
	IF AlarmCmdResetDevices THEN
		PT_Alarm.Cmd.ResetDevices := TRUE;
		AlarmCmdResetDevices := FALSE;
	END_IF;
	IF AlarmCmdResetProcess THEN
		PT_Alarm.Cmd.ResetProcess := TRUE;
		AlarmCmdResetProcess := FALSE;
	END_IF;

	AlarmAnyActive := PT_Alarm.Summary.AnyActive;
	AlarmAnyLatched := PT_Alarm.Summary.AnyLatched;
	AlarmAnyUnacknowledged := PT_Alarm.Summary.AnyUnacknowledged;
	AlarmAnyTrip := PT_Alarm.Summary.AnyTrip;
	AlarmRestartBlocked := PT_Alarm.Summary.RestartBlocked;
	AlarmHighestSeverity := PT_Alarm.Summary.HighestSeverity;
	AlarmFirstOutCode := PT_Alarm.Summary.FirstOutCode;
	AlarmActiveCount := PT_Alarm.Summary.ActiveCount;
	AlarmLatchedCount := PT_Alarm.Summary.LatchedCount;
	Alarm_21001 := PT_Alarm.Comm.BRB2.Latched;
	Alarm_21002 := PT_Alarm.Comm.IEBKB1.Latched;
	Alarm_21003 := PT_Alarm.Comm.BRB2RemoteFault.Latched;
	Alarm_22001 := PT_Alarm.Drive.PG_Pu01_VFD.Latched;
	Alarm_22002 := PT_Alarm.Drive.PG_Pu01_CAN.Latched;
	Alarm_22003 := PT_Alarm.Drive.PG_Pu02_VFD.Latched;
	Alarm_22004 := PT_Alarm.Drive.PG_Pu02_CAN.Latched;
	Alarm_25010 := PT_Alarm.Process.ValveRequestConflict.Latched;
	Alarm_25011 := PT_Alarm.Process.V01CloseTimeout.Latched;
	Alarm_25012 := PT_Alarm.Process.V02OpenTimeout.Latched;
	Alarm_25013 := PT_Alarm.Process.V02CloseTimeout.Latched;
	Alarm_25014 := PT_Alarm.Process.V01OpenTimeout.Latched;
	Alarm_25015 := PT_Alarm.Process.V01CloseIEBStopTimeout.Latched;
	Alarm_25016 := PT_Alarm.Process.IEBFlowStopTimeout.Latched;
	Alarm_25017 := PT_Alarm.Process.V05CloseTimeout.Latched;
	Alarm_25018 := PT_Alarm.Process.IEBFlowStartTimeout.Latched;
	Alarm_25021 := PT_Alarm.Process.BRB2FlowNotConfirmed.Latched;
	Alarm_25022 := PT_Alarm.Process.BRB2TemperatureNotReached.Latched;
	Alarm_25023 := PT_Alarm.Process.PT06HighPressure.Latched;
	Alarm_25031 := PT_Alarm.Process.TransferIEBFlowNotZero.Latched;
	Alarm_25032 := PT_Alarm.Process.TransferV05CloseTimeout.Latched;
	Alarm_25033 := PT_Alarm.Process.TransferV01CloseTimeout.Latched;
	Alarm_25034 := PT_Alarm.Process.TransferV02OpenTimeout.Latched;
	Alarm_25035 := PT_Alarm.Process.TransferBRB2FlowNotConfirmed.Latched;
	Alarm_26001 := PT_Alarm.AirRelease.PG_PV03.Latched;
	Alarm_26002 := PT_Alarm.AirRelease.PG_PV04.Latched;
	Alarm_41001 := PT_Alarm.IO.X20AI4622.Latched;
	Alarm_41002 := PT_Alarm.IO.X20AI4622a.Latched;
	Alarm_41003 := PT_Alarm.IO.X20AI4622b.Latched;
	Alarm_41004 := PT_Alarm.IO.X20AI4622c.Latched;
	Alarm_41005 := PT_Alarm.IO.X20AI4622d.Latched;
	Alarm_41101 := PT_Alarm.IO.X20AO4622.Latched;
	Alarm_41102 := PT_Alarm.IO.X20AO4622a.Latched;
	Alarm_41103 := PT_Alarm.IO.X20AO4622b.Latched;
	Alarm_41201 := PT_Alarm.IO.X20DI9371.Latched;
	Alarm_41202 := PT_Alarm.IO.X20DI9371a.Latched;
	Alarm_41203 := PT_Alarm.IO.X20DI9371b.Latched;
	Alarm_41301 := PT_Alarm.IO.X20DO9322.Latched;
	Alarm_41302 := PT_Alarm.IO.X20DO9322a.Latched;
	Alarm_41401 := PT_Alarm.IO.X20BC0083.Latched;
	Alarm_41402 := PT_Alarm.IO.X20PS9400.Latched;
	Alarm_41403 := PT_Alarm.IO.X20BT9100a.Latched;
	Alarm_41501 := PT_Alarm.IO.X67AI1323.Latched;
	Alarm_41502 := PT_Alarm.IO.X67AI1333b.Latched;
	Alarm_41601 := PT_Alarm.IO.X67DI1371_L12.Latched;
	Alarm_41701 := PT_Alarm.IO.X67DM1321_L12.Latched;
END_PROGRAM
```

#### Variables.var - Local variables
```iecst
VAR
	TrendClock : DTGetTime; (* Sistemsko vreme za granice 10-dnevnog trend zapisa. *)
	TrendNow_s : UDINT; (* Trenutno sistemsko vreme u sekundama od epohe. *)
	TrendEarliest_s : UDINT; (* Najstarije dostupno vreme unutar 10-dnevnog buffera. *)
	AlarmCmdAcknowledge : BOOL; (* HMI impuls za potvrdu svih alarma. *)
	AlarmCmdResetRecords : BOOL; (* HMI impuls za brisanje dozvoljenih alarmnih zapisa. *)
	AlarmCmdResetDevices : BOOL; (* HMI impuls za reset uredjaja bez procesnog starta. *)
	AlarmCmdResetProcess : BOOL; (* HMI impuls za reset procesa bez ponovnog starta. *)
	AlarmAnyActive : BOOL; (* Najmanje jedan alarmni uzrok je aktivan. *)
	AlarmAnyLatched : BOOL; (* Najmanje jedan alarm je memorisan. *)
	AlarmAnyUnacknowledged : BOOL; (* Najmanje jedan alarm nije potvrden. *)
	AlarmAnyTrip : BOOL; (* Najmanje jedan TRIP alarm postoji. *)
	AlarmRestartBlocked : BOOL; (* Novi procesni start je blokiran. *)
	AlarmHighestSeverity : USINT; (* Najvisi trenutni prioritet alarma. *)
	AlarmFirstOutCode : UINT; (* Kod prvog memorisanog alarma. *)
	AlarmActiveCount : UINT; (* Broj aktivnih alarmnih uzroka. *)
	AlarmLatchedCount : UINT; (* Broj memorisanih alarma. *)
	Alarm_21001 : BOOL;
	Alarm_21002 : BOOL;
	Alarm_21003 : BOOL;
	Alarm_22001 : BOOL;
	Alarm_22002 : BOOL;
	Alarm_22003 : BOOL;
	Alarm_22004 : BOOL;
	Alarm_25010 : BOOL;
	Alarm_25011 : BOOL;
	Alarm_25012 : BOOL;
	Alarm_25013 : BOOL;
	Alarm_25014 : BOOL;
	Alarm_25015 : BOOL;
	Alarm_25016 : BOOL;
	Alarm_25017 : BOOL;
	Alarm_25018 : BOOL;
	Alarm_25021 : BOOL;
	Alarm_25022 : BOOL;
	Alarm_25023 : BOOL;
	Alarm_25031 : BOOL;
	Alarm_25032 : BOOL;
	Alarm_25033 : BOOL;
	Alarm_25034 : BOOL;
	Alarm_25035 : BOOL;
	Alarm_26001 : BOOL;
	Alarm_26002 : BOOL;
	Alarm_41001 : BOOL; (* PT X20AI4622 module fault. *)
	Alarm_41002 : BOOL; (* PT X20AI4622a module fault. *)
	Alarm_41003 : BOOL; (* PT X20AI4622b module fault. *)
	Alarm_41004 : BOOL; (* PT X20AI4622c module fault. *)
	Alarm_41005 : BOOL; (* PT X20AI4622d module fault. *)
	Alarm_41101 : BOOL; (* PT X20AO4622 module fault. *)
	Alarm_41102 : BOOL; (* PT X20AO4622a module fault. *)
	Alarm_41103 : BOOL; (* PT X20AO4622b module fault. *)
	Alarm_41201 : BOOL; (* PT X20DI9371 module fault. *)
	Alarm_41202 : BOOL; (* PT X20DI9371a module fault. *)
	Alarm_41203 : BOOL; (* PT X20DI9371b module fault. *)
	Alarm_41301 : BOOL; (* PT X20DO9322 module fault. *)
	Alarm_41302 : BOOL; (* PT X20DO9322a module fault. *)
	Alarm_41401 : BOOL; (* PT X20BC0083 module fault. *)
	Alarm_41402 : BOOL; (* PT X20PS9400 module fault. *)
	Alarm_41403 : BOOL; (* PT X20BT9100a module fault. *)
	Alarm_41501 : BOOL; (* PT X67AI1323 module fault. *)
	Alarm_41502 : BOOL; (* PT X67AI1333b module fault. *)
	Alarm_41601 : BOOL; (* PT X67DI1371.L12 module fault. *)
	Alarm_41701 : BOOL; (* PT X67DM1321.L12 module fault. *)
END_VAR
```

- Visualisation Logical/Project/PG1_1 (not shown)

### Program Logical/Project/PID_Pu_PT (IEC)

#### Cyclic.st
```iecst
PROGRAM _CYCLIC
	(* ======================================================================== *)
	(* PID_PU_PT - REGULACIJA IZLAZNIH PUMPI PRIHVATNOG TANKA                *)
	(* AUTO: PID komande i frekvencija dolaze iz PGRad_Cmd.                   *)
	(* MANUAL: kada PGRad_Cmd nije aktivan, izlazne pumpe vode lokalne komande. *)
	(* STOP/FAULT: Disable PID i zaustavljanje izlaza imaju prioritet.         *)
	(* STATUS: UpdateDone i ostvarena frekvencija ostaju dostupni HMI-ju.      *)
	(* ======================================================================== *)
	(* ======================================================================== *)
	(* PID_Pu_PT_CYCLIC                                                           *)
	(* PID petlja pumpi na izlazu iz prihvatnog tanka.                            *)
	(* ======================================================================== *)

	(* -------------------------------------------------------------------------- *)
	(* 1) Rad po komandi state masine: PID je jedini vlasnik frekvencije i Run-a. *)
	(* -------------------------------------------------------------------------- *)
	(* Donja granica PID izlaza centralno se preuzima iz parametara pumpi. *)
	PID_Pu_PT.MinOut := PGRad.Par.MinFR_Pumpe;

	IF PGRad_Cmd.Aktivan THEN
		(* 1.1) Prenos procesnog zahteva u PID regulator. *)
		PID_Pu_PT.Enable := PGRad_Cmd.PID.Enable;
		PID_Pu_PT.ActValue := PGRad_Cmd.PID.ActValue;
		PID_Pu_PT.SetValue := PGRad_Cmd.PID.SetValue;
		PID_Pu_PT.Invert := PGRad_Cmd.PID.Invert;
		PID_Pu_PT.MaxOut := PGRad_Cmd.PID.MaxOut; (* Preuzima PGRad.Par.MaxFR_Pumpe. *)
		PID_Pu_PT.EnableTracking := PGRad_Cmd.PID.EnableTracking;
		PID_Pu_PT.TrackingValue := PGRad_Cmd.PID.TrackingValue;
		IF EDGEPOS(PGRad_Cmd.PID.Enable) THEN
			PID_Pu_PT.Update := TRUE;
		END_IF
		PID_Pu_PT();
		IF PID_Pu_PT.UpdateDone THEN
			PID_Pu_PT.Update := FALSE;
		END_IF

		(* 1.2) Iskljucivo izabrana izlazna pumpa dobija PID frekvenciju i Run. *)
		PG.Act.Pu._1.Start := FALSE;
		PG.Act.Pu._2.Start := FALSE;
		IF PGRad_Cmd.PID.Enable THEN
			IF PGRad_Cmd.Pumpe._01.Run THEN
				PG.Act.Pu._1.FR_set := PID_Pu_PT.Out;
				PG.Act.Pu._1.Start := TRUE;
			ELSIF PGRad_Cmd.Pumpe._02.Run THEN
				PG.Act.Pu._2.FR_set := PID_Pu_PT.Out;
				PG.Act.Pu._2.Start := TRUE;
			END_IF
		END_IF

	ELSE
		(* -------------------------------------------------------------------------- *)
		(* 2) Rucni rad pumpi                                                       *)
		(* -------------------------------------------------------------------------- *)
		(* U rucnom rezimu HMI neposredno zadaje Start i FR_set izabrane pumpe. *)
		PID_Pu_PT.Enable := FALSE;
		PID_Pu_PT.EnableTracking := FALSE;
		PID_Pu_PT();

		(* -------------------------------------------------------------------------- *)
		(* 3) Zadrzavanje postojeceg nasledjenog bypass zahteva                     *)
		(* -------------------------------------------------------------------------- *)
		(* PG_V05 prati otvoren ulazni ventil PG_V01 u nasledjenom lokalnom rezimu. *)
		IF PG.Act.AV._1.Open THEN
			PG.Act.AV._5.Open := TRUE;
		END_IF
	END_IF
END_PROGRAM
```

#### Init.st
```iecst
PROGRAM _INIT
	(* ======================================================================== *)
	(* PID_Pu_PT_INIT                                                             *)
	(* PID petlja pumpi na izlazu iz prihvatnog tanka.                            *)
	(* Procesni rezim kasnije prosledjuje aktivne PV/SP, smer i izlazne granice. *)
	(* ======================================================================== *)
	(* -------------------------------------------------------------------------- *)
	(* 1) Inicijalni parametri PID izlazne pumpe                                  *)
	(* -------------------------------------------------------------------------- *)
	(* Granice PID izlaza preuzimaju se iz centralnih parametara pumpi. *)
	PID_Pu_PT.MaxOut := PGRad.Par.MaxFR_Pumpe; (* Gornja granica iz MaxFR_Pumpe [Hz]. *)
	PID_Pu_PT.MinOut := PGRad.Par.MinFR_Pumpe; (* Donja granica iz MinFR_Pumpe [Hz]. *)

	(* Parametri nivo regulacije; D clan je iskljucen. *)
	(* FilterTime filtrira D clan i nema uticaja dok je DerivativeTime = 0.0. *)
	PID_Pu_PT.PIDParameters.DerivativeTime := 0.0; (* D vreme [s]. *)
	PID_Pu_PT.PIDParameters.FilterTime := 10.0; (* Vremenska konstanta filtera D clana [s]. *)
	PID_Pu_PT.PIDParameters.Gain := 96.3; (* Proporcionalno pojacanje. *)
	PID_Pu_PT.PIDParameters.IntegrationTime := 180; (* Integraciono vreme [s]. *)
	PID_Pu_PT.Invert := TRUE; (* Nivo regulacija koristi inverzni smer. *)

	PID_Pu_PT.SetValue := 1.5; (* Lokalni pocetni setpoint nivoa [m]. *)

END_PROGRAM
```

### Program Logical/Project/AlarmMgr (IEC)

#### Init.st - Init code
```iecst
PROGRAM _INIT
	(* ======================================================================== *)
	(* 1) Neretentivno pocetno stanje alarmnog sistema                          *)
	(* ======================================================================== *)
	PT_Alarm.Cmd.AcknowledgeAll := FALSE;
	PT_Alarm.Cmd.ResetAlarmRecords := FALSE;
	PT_Alarm.Cmd.ResetDevices := FALSE;
	PT_Alarm.Cmd.ResetProcess := FALSE;
	PT_Alarm.ResetPulse.Devices := FALSE;
	PT_Alarm.ResetPulse.Process := FALSE;
	PT_Alarm.Summary.FirstOutCode := 0;

	(* ======================================================================== *)
	(* 2) Stabilni kodovi, prioriteti i blokade                                 *)
	(* ======================================================================== *)
	PT_Alarm.Comm.BRB2.Code := 21001;
	PT_Alarm.Comm.BRB2.Severity := 4;
	PT_Alarm.Comm.BRB2.Blocking := TRUE;
	PT_Alarm.Comm.IEBKB1.Code := 21002;
	PT_Alarm.Comm.IEBKB1.Severity := 4;
	PT_Alarm.Comm.IEBKB1.Blocking := TRUE;
	PT_Alarm.Comm.BRB2RemoteFault.Code := 21003;
	PT_Alarm.Comm.BRB2RemoteFault.Severity := 4;
	PT_Alarm.Comm.BRB2RemoteFault.Blocking := TRUE;

	PT_Alarm.Drive.PG_Pu01_VFD.Code := 22001;
	PT_Alarm.Drive.PG_Pu01_VFD.Severity := 4;
	PT_Alarm.Drive.PG_Pu01_VFD.Blocking := TRUE;
	PT_Alarm.Drive.PG_Pu01_CAN.Code := 22002;
	PT_Alarm.Drive.PG_Pu01_CAN.Severity := 4;
	PT_Alarm.Drive.PG_Pu01_CAN.Blocking := TRUE;
	PT_Alarm.Drive.PG_Pu02_VFD.Code := 22003;
	PT_Alarm.Drive.PG_Pu02_VFD.Severity := 4;
	PT_Alarm.Drive.PG_Pu02_VFD.Blocking := TRUE;
	PT_Alarm.Drive.PG_Pu02_CAN.Code := 22004;
	PT_Alarm.Drive.PG_Pu02_CAN.Severity := 4;
	PT_Alarm.Drive.PG_Pu02_CAN.Blocking := TRUE;

	PT_Alarm.Process.ValveRequestConflict.Code := 25010;
	PT_Alarm.Process.ValveRequestConflict.SourceCode := 10;
	PT_Alarm.Process.V01CloseTimeout.Code := 25011;
	PT_Alarm.Process.V01CloseTimeout.SourceCode := 11;
	PT_Alarm.Process.V02OpenTimeout.Code := 25012;
	PT_Alarm.Process.V02OpenTimeout.SourceCode := 12;
	PT_Alarm.Process.V02CloseTimeout.Code := 25013;
	PT_Alarm.Process.V02CloseTimeout.SourceCode := 13;
	PT_Alarm.Process.V01OpenTimeout.Code := 25014;
	PT_Alarm.Process.V01OpenTimeout.SourceCode := 14;
	PT_Alarm.Process.V01CloseIEBStopTimeout.Code := 25015;
	PT_Alarm.Process.V01CloseIEBStopTimeout.SourceCode := 15;
	PT_Alarm.Process.IEBFlowStopTimeout.Code := 25016;
	PT_Alarm.Process.IEBFlowStopTimeout.SourceCode := 16;
	PT_Alarm.Process.V05CloseTimeout.Code := 25017;
	PT_Alarm.Process.V05CloseTimeout.SourceCode := 17;
	PT_Alarm.Process.IEBFlowStartTimeout.Code := 25018;
	PT_Alarm.Process.IEBFlowStartTimeout.SourceCode := 18;
	PT_Alarm.Process.BRB2FlowNotConfirmed.Code := 25021;
	PT_Alarm.Process.BRB2FlowNotConfirmed.SourceCode := 21;
	PT_Alarm.Process.BRB2TemperatureNotReached.Code := 25022;
	PT_Alarm.Process.BRB2TemperatureNotReached.SourceCode := 22;
	PT_Alarm.Process.PT06HighPressure.Code := 25023;
	PT_Alarm.Process.PT06HighPressure.SourceCode := 23;
	PT_Alarm.Process.TransferIEBFlowNotZero.Code := 25031;
	PT_Alarm.Process.TransferIEBFlowNotZero.SourceCode := 31;
	PT_Alarm.Process.TransferV05CloseTimeout.Code := 25032;
	PT_Alarm.Process.TransferV05CloseTimeout.SourceCode := 32;
	PT_Alarm.Process.TransferV01CloseTimeout.Code := 25033;
	PT_Alarm.Process.TransferV01CloseTimeout.SourceCode := 33;
	PT_Alarm.Process.TransferV02OpenTimeout.Code := 25034;
	PT_Alarm.Process.TransferV02OpenTimeout.SourceCode := 34;
	PT_Alarm.Process.TransferBRB2FlowNotConfirmed.Code := 25035;
	PT_Alarm.Process.TransferBRB2FlowNotConfirmed.SourceCode := 35;

	PT_Alarm.Process.ValveRequestConflict.Severity := 4;
	PT_Alarm.Process.V01CloseTimeout.Severity := 4;
	PT_Alarm.Process.V02OpenTimeout.Severity := 4;
	PT_Alarm.Process.V02CloseTimeout.Severity := 4;
	PT_Alarm.Process.V01OpenTimeout.Severity := 4;
	PT_Alarm.Process.V01CloseIEBStopTimeout.Severity := 4;
	PT_Alarm.Process.IEBFlowStopTimeout.Severity := 4;
	PT_Alarm.Process.V05CloseTimeout.Severity := 4;
	PT_Alarm.Process.IEBFlowStartTimeout.Severity := 4;
	PT_Alarm.Process.BRB2FlowNotConfirmed.Severity := 4;
	PT_Alarm.Process.BRB2TemperatureNotReached.Severity := 4;
	PT_Alarm.Process.PT06HighPressure.Severity := 4;
	PT_Alarm.Process.TransferIEBFlowNotZero.Severity := 4;
	PT_Alarm.Process.TransferV05CloseTimeout.Severity := 4;
	PT_Alarm.Process.TransferV01CloseTimeout.Severity := 4;
	PT_Alarm.Process.TransferV02OpenTimeout.Severity := 4;
	PT_Alarm.Process.TransferBRB2FlowNotConfirmed.Severity := 4;

	PT_Alarm.Process.ValveRequestConflict.Blocking := TRUE;
	PT_Alarm.Process.V01CloseTimeout.Blocking := TRUE;
	PT_Alarm.Process.V02OpenTimeout.Blocking := TRUE;
	PT_Alarm.Process.V02CloseTimeout.Blocking := TRUE;
	PT_Alarm.Process.V01OpenTimeout.Blocking := TRUE;
	PT_Alarm.Process.V01CloseIEBStopTimeout.Blocking := TRUE;
	PT_Alarm.Process.IEBFlowStopTimeout.Blocking := TRUE;
	PT_Alarm.Process.V05CloseTimeout.Blocking := TRUE;
	PT_Alarm.Process.IEBFlowStartTimeout.Blocking := TRUE;
	PT_Alarm.Process.BRB2FlowNotConfirmed.Blocking := TRUE;
	PT_Alarm.Process.BRB2TemperatureNotReached.Blocking := TRUE;
	PT_Alarm.Process.PT06HighPressure.Blocking := TRUE;
	PT_Alarm.Process.TransferIEBFlowNotZero.Blocking := TRUE;
	PT_Alarm.Process.TransferV05CloseTimeout.Blocking := TRUE;
	PT_Alarm.Process.TransferV01CloseTimeout.Blocking := TRUE;
	PT_Alarm.Process.TransferV02OpenTimeout.Blocking := TRUE;
	PT_Alarm.Process.TransferBRB2FlowNotConfirmed.Blocking := TRUE;

	PT_Alarm.AirRelease.PG_PV03.Code := 26001;
	PT_Alarm.AirRelease.PG_PV03.Severity := 3;
	PT_Alarm.AirRelease.PG_PV03.Blocking := FALSE;
	PT_Alarm.AirRelease.PG_PV04.Code := 26002;
	PT_Alarm.AirRelease.PG_PV04.Severity := 3;
	PT_Alarm.AirRelease.PG_PV04.Blocking := FALSE;
END_PROGRAM
```
